(* CODESYS project Struckig_0.17.3.2.library
   Company: Stefan Besler
   DefaultNamespace: Struckig
   Version: 0.17.3.2
   Placeholder: Struckig
   Author: Stefan Besler and contributers
   Description: Full port of pantor ruckig library (Community version) to IEC 61131-3 Structured Text. Online Trajectory Generation. Real-time. Time-optimal. Jerk-constrained.
   Title: Struckig

Project tree, tasks and I/O mapping:
  Struckig/
    _DataTypes/
      data type ControlInterfaceType
      data type DiscretizationType
      data type SynchronizationType
      data type TrajectoryErrorCode
      data type TrajectoryState
    Block/
      data type Block
      data type BlockInterval
    BrakeProfile/
      function block BrakeProfile [ST]: AccelerationBrake, Finalize, FinalizeSecondOrder, PositionBrakeTrajectory, SecondOrderPositionBrakeTrajectory, SecondOrderVelocityBrakeTrajectory, SmoothVelocityBrake, VelocityAtTime, VelocityAtZeroAcceleration, velocityBrake, VelocityBrakeTrajectory
    Math/
      function BubbleSortLreal [ST]
      function Cbrt [ST]
      function Ceil [ST]
      function Clamp [ST]
      function Fmod [ST]
      function IsInfinity [ST]
      function IsNaN [ST]
      function LrealBits [ST]
      function LrealFromBits [ST]
      function Power [ST]
      function Power2 [ST]
      program Roots [ST]: PolyDeri, PolyEval, PolyMonicDeri, ShrinkInterval, SolveCub, SolveQuartMonic, SolveResolvent
    Position/
      function block PositionFirstOrderStep1 [ST]: Get, Set
      function block PositionFirstOrderStep2 [ST]: Get, Set
      function block PositionSecondOrderStep1 [ST]: AddInterval, AddProfile, CalculateBlock, Get, RemoveProfile, Set, time_acc0, time_all_single_step, time_none
      function block PositionSecondOrderStep2 [ST]: CheckAll, Get, Set, time_acc0, time_none
      function block PositionThirdOrderStep1 [ST]: AddInterval, AddProfile, CalculateBlock, Get, RemoveProfile, Set, time_acc0_acc1, time_acc0_two_step, time_acc1_vel_two_step, time_all_none_acc0_acc1, time_all_single_step, time_all_vel, time_none_two_step, time_vel_two_step
      function block PositionThirdOrderStep2 [ST]: Get, Set, time_acc0, time_acc0_acc1, time_acc0_acc1_vel, time_acc0_vel, time_acc1, time_acc1_vel, time_none, time_none_smooth, time_vel
    Profile/
      _DataTypes/
        data type ProfileBound
        data type ProfileControlSigns
        data type ProfileDirection
        data type ReachedLimits
      function block ProfileDesc [ST]: Bound, CheckBound, CheckForFirstOrder, CheckForFirstOrderWithTiming, CheckForFirstOrderWithTiming2, CheckForSecondOrder, CheckForSecondOrderVelocity, CheckForSecondOrderVelocityWithTiming, CheckForSecondOrderVelocityWithTiming2, CheckForSecondOrderWithTiming, CheckForSecondOrderWithTiming2, CheckForVelocity, CheckForVelocityWithTiming, CheckStepForBound, CheckVel, CheckWithTiming, CheckWithTiming2, FirstStateAtPosition, SetBoundary, SetBoundaryPosition, SetBoundaryVelocity
    Velocity/
      function block VelocitySecondOrderStep1 [ST]: Get, Set
      function block VelocitySecondOrderStep2 [ST]: Get, Set
      function block VelocityThirdOrderStep1 [ST]: AddInterval, AddProfile, CalculateBlock, Get, RemoveProfile, Set, time_acc0, time_all_single_step, time_none
      function block VelocityThirdOrderStep2 [ST]: CheckAll, Get, Set, time_acc0, time_none
    function Integrate [ST]
    interface IOtg: AtTime, AtTime1, Cyclic, Duration, ErrorCode, ErrorMessage, PassOutputToInput, Reset, State, ValidateInput
    function block Otg [ST]: AbortErrorId, AtTime, AtTime1, Calculate, Cyclic, Duration, ErrorCode, ErrorMessage, FB_init, HasChanged, IsBlocked, IsInputCollinear, PassOutputToInput, Reset, SetBusy, State, Synchronize, ValidateInput, ValidateInputOrAbort, VelocityAtZero
    function block Otg1 [ST]: AtTime, AtTime1, Cyclic, Duration, ErrorCode, ErrorMessage, FB_init, PassOutputToInput, Reset, State, ValidateInput
  global variables Constants
  global variables ParameterList
*)

// Struckig/_DataTypes/ControlInterfaceType
// Struckig
// Copyright (C) 2022 Stefan Besler

// This program is free software: you can redistribute it and/or modify
// it under the terms of the GNU General Public License as published by
// the Free Software Foundation, either version 3 of the License, or
// (at your option) any later version.

// This program is distributed in the hope that it will be useful,
// but WITHOUT ANY WARRANTY; without even the implied warranty of
// MERCHANTABILITY or FITNESS FOR A PARTICULAR PURPOSE.  See the
// GNU General Public License for more details.
//
// You should have received a copy of the GNU General Public License
// along with THIS PROGRAM.  IF NOT, see <http://www.gnu.org/licenses/>.
{attribute 'qualified_only'}
{attribute 'strict'}
/// Defines the controlled state variables for trajectory generation.
/// The selected mode changes which boundary values and limits are interpreted
/// during validation and profile generation.
TYPE ControlInterfaceType :
(
  Undefined, //< Use global/default configuration.
  Position, //< Full control over position, velocity, and acceleration.
  Velocity //< Controls only velocity and acceleration states.
);
END_TYPE

// Struckig/_DataTypes/DiscretizationType
// Struckig
// Copyright (C) 2022 Stefan Besler

// This program is free software: you can redistribute it and/or modify
// it under the terms of the GNU General Public License as published by
// the Free Software Foundation, either version 3 of the License, or
// (at your option) any later version.

// This program is distributed in the hope that it will be useful,
// but WITHOUT ANY WARRANTY; without even the implied warranty of
// MERCHANTABILITY or FITNESS FOR A PARTICULAR PURPOSE.  See the
// GNU General Public License for more details.
//
// You should have received a copy of the GNU General Public License
// along with THIS PROGRAM.  IF NOT, see <http://www.gnu.org/licenses/>.
{attribute 'qualified_only'}
{attribute 'strict'}
/// Defines whether synchronized trajectory duration is continuous or cycle-discrete.
TYPE DiscretizationType :
(
  Continuous, //< Every synchronization duration is allowed.
  Discrete //< Synchronization duration must be a multiple of cycle time.
);
END_TYPE

// Struckig/_DataTypes/SynchronizationType
// Struckig
// Copyright (C) 2022 Stefan Besler

// This program is free software: you can redistribute it and/or modify
// it under the terms of the GNU General Public License as published by
// the Free Software Foundation, either version 3 of the License, or
// (at your option) any later version.

// This program is distributed in the hope that it will be useful,
// but WITHOUT ANY WARRANTY; without even the implied warranty of
// MERCHANTABILITY or FITNESS FOR A PARTICULAR PURPOSE.  See the
// GNU General Public License for more details.
//
// You should have received a copy of the GNU General Public License
// along with THIS PROGRAM.  IF NOT, see <http://www.gnu.org/licenses/>.
{attribute 'qualified_only'}
{attribute 'strict'}
/// Defines how multiple DoFs are synchronized to a common trajectory timing.
/// This setting is evaluated together with per-axis overrides (`PerDofSynchronization`)
/// in [Otg](xref:Struckig.Otg).
TYPE SynchronizationType :
(
  Undefined, //< Use global/default configuration.
  TimeSync, //< Always synchronize the DoFs to reach the target at the same time (Default)
  TimeIfNecessarySync, //< Synchronize only when necessary (e.g. for non-zero target velocity or acceleration)
  Phase,  //< Phase synchronize the DoFs when this is possible, else fallback to "Time" strategy. Phase synchronization will result a straight-line trajectory
    // PhaseOnly, //< Always phase synchronize the DoFs (even when this is not time-optimal), else returns "ErrorNoPhaseSynchronization". Ruckig will then guarantee a straight-line trajectory
  None //< Calculate every DoF independently
);
END_TYPE

// Struckig/_DataTypes/TrajectoryErrorCode
// Struckig
// Copyright (C) 2022 Stefan Besler

// This program is free software: you can redistribute it and/or modify
// it under the terms of the GNU General Public License as published by
// the Free Software Foundation, either version 3 of the License, or
// (at your option) any later version.

// This program is distributed in the hope that it will be useful,
// but WITHOUT ANY WARRANTY; without even the implied warranty of
// MERCHANTABILITY or FITNESS FOR A PARTICULAR PURPOSE.  See the
// GNU General Public License for more details.
//
// You should have received a copy of the GNU General Public License
// along with THIS PROGRAM.  IF NOT, see <http://www.gnu.org/licenses/>.
{attribute 'qualified_only'}
/// Error codes reported by the trajectory generator.
/// Returned by [ErrorCode](xref:Struckig.IOtg#ErrorCode) and explained by
/// [ErrorMessage](xref:Struckig.IOtg#ErrorMessage).
TYPE TrajectoryErrorCode :
(
  Undefined := 0, //< No error.
  InvalidInput, //< Error in the input parameter
  SynchronizationFailed, //< No valid synchronized profile was found.
  CalculateStep1Failed, //< Profile search in step 1 failed.
  ZeroLimitsConflict, //< Conflicting zero limits prevent profile generation.
  ZeroLimitsConflictInSynchronization //< Zero-limit conflict during multi-DoF synchronization.
);
END_TYPE

// Struckig/_DataTypes/TrajectoryState
// Struckig
// Copyright (C) 2022 Stefan Besler

// This program is free software: you can redistribute it and/or modify
// it under the terms of the GNU General Public License as published by
// the Free Software Foundation, either version 3 of the License, or
// (at your option) any later version.

// This program is distributed in the hope that it will be useful,
// but WITHOUT ANY WARRANTY; without even the implied warranty of
// MERCHANTABILITY or FITNESS FOR A PARTICULAR PURPOSE.  See the
// GNU General Public License for more details.
//
// You should have received a copy of the GNU General Public License
// along with THIS PROGRAM.  IF NOT, see <http://www.gnu.org/licenses/>.
{attribute 'qualified_only'}
{attribute 'strict'}
/// Runtime state of the trajectory generator.
TYPE TrajectoryState :
(
  Undefined, //< State has not been initialized yet.
  
  /// The trajectory has reached its final position. For trajectories with a target velocity or/and a target acceleration
  /// there will still be movement.
  Idle,
  
  /// The trajectory is calculated normally
  Busy,
  
  /// An error occured, use [ErrorCode](xref:Struckig.IOtg#ErrorCode) and [ErrorMessage](xref:Struckig.IOtg#ErrorMessage) to get more
  /// information about the error.
  Error
);
END_TYPE

// Struckig/Block/Block
// Struckig
// Copyright (C) 2022 Stefan Besler

// This program is free software: you can redistribute it and/or modify
// it under the terms of the GNU General Public License as published by
// the Free Software Foundation, either version 3 of the License, or
// (at your option) any later version.

// This program is distributed in the hope that it will be useful,
// but WITHOUT ANY WARRANTY; without even the implied warranty of
// MERCHANTABILITY or FITNESS FOR A PARTICULAR PURPOSE.  See the
// GNU General Public License for more details.
//
// You should have received a copy of the GNU General Public License
// along with THIS PROGRAM.  IF NOT, see <http://www.gnu.org/licenses/>.
TYPE INTERNAL Block :
STRUCT
  Pmin : ProfileDesc; // Save min Profile so that it doesn't need to be recalculated in Step2
  Tmin : LREAL; // [s]
  A, B : BlockInterval; // Max. 2 intervals can be blocked: called a and b with corresponding profiles, order does not matter  
END_STRUCT
END_TYPE

// Struckig/Block/BlockInterval
// Struckig
// Copyright (C) 2022 Stefan Besler

// This program is free software: you can redistribute it and/or modify
// it under the terms of the GNU General Public License as published by
// the Free Software Foundation, either version 3 of the License, or
// (at your option) any later version.

// This program is distributed in the hope that it will be useful,
// but WITHOUT ANY WARRANTY; without even the implied warranty of
// MERCHANTABILITY or FITNESS FOR A PARTICULAR PURPOSE.  See the
// GNU General Public License for more details.
//
// You should have received a copy of the GNU General Public License
// along with THIS PROGRAM.  IF NOT, see <http://www.gnu.org/licenses/>.
/// Which times are possible for synchronization?
TYPE INTERNAL BlockInterval :
STRUCT
  IsUsed : BOOL;
  Left, Right : LREAL;
  Profile : ProfileDesc;
END_STRUCT
END_TYPE

// Struckig/Profile/_DataTypes/ProfileBound
// Struckig
// Copyright (C) 2022 Stefan Besler

// This program is free software: you can redistribute it and/or modify
// it under the terms of the GNU General Public License as published by
// the Free Software Foundation, either version 3 of the License, or
// (at your option) any later version.

// This program is distributed in the hope that it will be useful,
// but WITHOUT ANY WARRANTY; without even the implied warranty of
// MERCHANTABILITY or FITNESS FOR A PARTICULAR PURPOSE.  See the
// GNU General Public License for more details.
//
// You should have received a copy of the GNU General Public License
// along with THIS PROGRAM.  IF NOT, see <http://www.gnu.org/licenses/>.
{attribute 'conditionalshow'}
/// Positional envelope of a single-DoF profile.
/// The structure stores minimum/maximum position and the corresponding
/// times where these extrema occur along the generated trajectory.
///
/// It is returned by profile-bound checks to answer questions such as:
/// "What is the furthest negative/positive excursion and when does it happen?"
TYPE ProfileBound :
STRUCT
  Minimum, Maximum : LREAL; //< Extreme positions reached by the profile.
  Tmin, Tmax : LREAL;  //< Times at which `Minimum` and `Maximum` are reached.
END_STRUCT
END_TYPE

// Struckig/Profile/_DataTypes/ProfileControlSigns
// Struckig
// Copyright (C) 2022 Stefan Besler

// This program is free software: you can redistribute it and/or modify
// it under the terms of the GNU General Public License as published by
// the Free Software Foundation, either version 3 of the License, or
// (at your option) any later version.

// This program is distributed in the hope that it will be useful,
// but WITHOUT ANY WARRANTY; without even the implied warranty of
// MERCHANTABILITY or FITNESS FOR A PARTICULAR PURPOSE.  See the
// GNU General Public License for more details.
//
// You should have received a copy of the GNU General Public License
// along with THIS PROGRAM.  IF NOT, see <http://www.gnu.org/licenses/>.
{attribute 'qualified_only'}
{attribute 'strict'}
TYPE INTERNAL ProfileControlSigns :
(
  Uddu,
  Udud 
);
END_TYPE

// Struckig/Profile/_DataTypes/ProfileDirection
// Struckig
// Copyright (C) 2022 Stefan Besler

// This program is free software: you can redistribute it and/or modify
// it under the terms of the GNU General Public License as published by
// the Free Software Foundation, either version 3 of the License, or
// (at your option) any later version.

// This program is distributed in the hope that it will be useful,
// but WITHOUT ANY WARRANTY; without even the implied warranty of
// MERCHANTABILITY or FITNESS FOR A PARTICULAR PURPOSE.  See the
// GNU General Public License for more details.
//
// You should have received a copy of the GNU General Public License
// along with THIS PROGRAM.  IF NOT, see <http://www.gnu.org/licenses/>.
{attribute 'qualified_only'}
{attribute 'strict'}
TYPE INTERNAL ProfileDirection :
(
  Up,
  Down
);
END_TYPE

// Struckig/Profile/_DataTypes/ReachedLimits
// Struckig
// Copyright (C) 2022 Stefan Besler

// This program is free software: you can redistribute it and/or modify
// it under the terms of the GNU General Public License as published by
// the Free Software Foundation, either version 3 of the License, or
// (at your option) any later version.

// This program is distributed in the hope that it will be useful,
// but WITHOUT ANY WARRANTY; without even the implied warranty of
// MERCHANTABILITY or FITNESS FOR A PARTICULAR PURPOSE.  See the
// GNU General Public License for more details.
//
// You should have received a copy of the GNU General Public License
// along with THIS PROGRAM.  IF NOT, see <http://www.gnu.org/licenses/>.
{attribute 'qualified_only'}
{attribute 'strict'}
TYPE INTERNAL ReachedLimits :
(
  Acc0Acc1Vel,
  Vel, 
  Acc0,
  Acc1,
  Acc0Acc1,
  Acc0Vel,
  Acc1Vel,
  None
);
END_TYPE

// Constants
// Struckig
// Copyright (C) 2022 Stefan Besler

// This program is free software: you can redistribute it and/or modify
// it under the terms of the GNU General Public License as published by
// the Free Software Foundation, either version 3 of the License, or
// (at your option) any later version.

// This program is distributed in the hope that it will be useful,
// but WITHOUT ANY WARRANTY; without even the implied warranty of
// MERCHANTABILITY or FITNESS FOR A PARTICULAR PURPOSE.  See the
// GNU General Public License for more details.
//
// You should have received a copy of the GNU General Public License
// along with THIS PROGRAM.  IF NOT, see <http://www.gnu.org/licenses/>.
{attribute 'qualified_only'}
{attribute 'hide'}
VAR_GLOBAL CONSTANT
  BrakeEpsilon : LREAL := 2.2E-14;
  DoubleEpsilon : LREAL := 2.2204460492503131E-016; // smallest such that 1.0+Constants.DoubleEpsilon != 1.0
  Epsilon : LREAL := 1E-8;
  Epsilon16 : LREAL := 16 * 2.2204460492503131E-016;
  EpsilonColinear : LREAL := 1E-7;
  Infinity : LREAL := 1.7976931348623157E+308;  
  Tolerance : LREAL := 1E-14;
  Cos120 : LREAL := -0.50;
  Sin120 : LREAL := 0.866025403784438646764;  
  Pi : LREAL := 3.14159265358979323846;
  Minimum : LREAL := 1.17549435082E-38;  // used for validating input
  
  VelocityEpsilon : LREAL := 1E-12;
  AccelerationEpsilon : LREAL := 1E-12;
  JerkEpsilon : LREAL := 1E-12; 
  
  PositionPrecision : LREAL := 1E-8;
  VelocityPrecision : LREAL := 1E-8;
  AccelerationPrecision : LREAL := 1E-10;
  TimePrecision : LREAL := 1E-12;  
  
  Tmax : LREAL := 1E12;
END_VAR

// ParameterList
// Struckig
// Copyright (C) 2022 Stefan Besler

// This program is free software: you can redistribute it and/or modify
// it under the terms of the GNU General Public License as published by
// the Free Software Foundation, either version 3 of the License, or
// (at your option) any later version.

// This program is distributed in the hope that it will be useful,
// but WITHOUT ANY WARRANTY; without even the implied warranty of
// MERCHANTABILITY or FITNESS FOR A PARTICULAR PURPOSE.  See the
// GNU General Public License for more details.
//
// You should have received a copy of the GNU General Public License
// along with THIS PROGRAM.  IF NOT, see <http://www.gnu.org/licenses/>.
{attribute 'qualified_only'}
/// Global configuration constants for Struckig.
/// These values define library limits and algorithm defaults that are
/// referenced by trajectory generation and numerical helper routines.
VAR_GLOBAL CONSTANT
  MaxDoFs : INT := 7; //< Maximum number of degrees of freedom supported by `Otg`.
  MaxIterations : BYTE := 127; //< Maximum iterations when [shrinking an interval](xref:Struckig.Roots#ShrinkInterval)
  NumericalRobust : BOOL := TRUE; //< Enables additional guards for numerically robust calculations.
  
  /// Default initial value for Otg.SmoothBrake / Otg1.SmoothBrake
  /// If enabled, braking profiles prefer smooth acceleration transitions.
  SmoothBrake : BOOL := FALSE;
END_VAR

// Struckig/BrakeProfile/BrakeProfile
// Struckig
// Copyright (C) 2022 Stefan Besler

// This program is free software: you can redistribute it and/or modify
// it under the terms of the GNU General Public License as published by
// the Free Software Foundation, either version 3 of the License, or
// (at your option) any later version.

// This program is distributed in the hope that it will be useful,
// but WITHOUT ANY WARRANTY; without even the implied warranty of
// MERCHANTABILITY or FITNESS FOR A PARTICULAR PURPOSE.  See the
// GNU General Public License for more details.
//
// You should have received a copy of the GNU General Public License
// along with THIS PROGRAM.  IF NOT, see <http://www.gnu.org/licenses/>.
/// Calculates (pre- or post-) profile to get current or final state below the limits
FUNCTION_BLOCK BrakeProfile
VAR_INPUT
  Duration : LREAL; //! Overall duration
  t, j, a, v, p : ARRAY[0..2] OF LREAL; //! Profile information for up to three-step profile  
  IsUsed : BOOL;
END_VAR
VAR
  t_to_a_min, t_to_a_max, t_min_to_v_max, t_to_a_zero, t_to_v_min, t_to_v_max : LREAL;
  t_to_v_max_with_constant, t_to_v_min_with_constant, v_at_a0, v_at_a_max, v_at_a_min : LREAL;
END_VAR

METHOD AccelerationBrake
VAR_INPUT
  v0, a0 : LREAL;
  vMax, vMin : LREAL;
  aMax, aMin : LREAL;
  jMax : LREAL;
END_VAR
j[0] := -jMax;

t_to_a_max := (a0 - aMax) / jMax;
t_to_a_zero := a0 / jMax;

v_at_a_max := VelocityAtTime(v0, a0, -jMax, t_to_a_max);
v_at_a0 := VelocityAtTime(v0, a0, -jMax, t_to_a_zero);

IF (v_at_a0 > vMax AND_THEN jMax > 0) OR_ELSE (v_at_a0 < vMax AND_THEN jMax < 0)
THEN
  VelocityBrake(v0, a0, vMax, vMin, aMax, aMin, jMax);

ELSIF (v_at_a_max < vMin AND_THEN jMax > 0) OR_ELSE (v_at_a_max > vMin AND_THEN jMax < 0)
THEN
  t_to_v_min := -(v_at_a_max - vMin)/aMax;
  t_to_v_max := -aMax/(2*jMax) - (v_at_a_max + vMax)/aMax;
  t[0] := t_to_a_max + Constants.BrakeEpsilon;
  t[1] := MAX(MIN(t_to_v_min, v_at_a_max - Constants.BrakeEpsilon), 0.0);
ELSE
  t[0] := t_to_a_max + Constants.BrakeEpsilon;
END_IF
END_METHOD

/// Finalize third-order braking by integrating along kinematic state
METHOD Finalize
VAR_IN_OUT
  ps : LREAL;
  vs : LREAL;
  as : LREAL;
END_VAR
IF t[0] <= 0 AND_THEN t[1] <= 0
THEN
  Duration := 0;
  RETURN;
END_IF

Duration := t[0];
p[0] := ps;
v[0] := vs;
a[0] := as;
Integrate(t[0], p0:=ps, v0:=vs, a0:=as, j:=j[0], p:=ps, v:=vs, a:=as);

IF t[1] > 0
THEN
  Duration := Duration + t[1];
  p[1] := ps;
  v[1] := vs;
  a[1] := as;
  Integrate(t[1], p0:=ps, v0:=vs, a0:=as, j:=j[1], p:=ps, v:=vs, a:=as);
END_IF

IF t[2] > 0
THEN
  Duration := Duration + t[2];
  p[2] := ps;
  v[2] := vs;
  a[2] := as;
  Integrate(t[2], p0:=ps, v0:=vs, a0:=as, j:=j[2], p:=ps, v:=vs, a:=as);
END_IF
END_METHOD

/// Finalize third-order braking by integrating along kinematic state
METHOD FinalizeSecondOrder
VAR_IN_OUT
  ps : LREAL;
  vs : LREAL;
  as : LREAL;
END_VAR
IF t[0] <= 0.0
THEN
  Duration := 0;
  RETURN;
END_IF

Duration := t[0];
p[0] := ps;
v[0] := vs;
Integrate(t[0], p0:=ps, v0:=vs, a0:=a[0], j:=j[0], p:=ps, v:=vs, a:=as);
END_METHOD

/// Calculate brake trajectory for third-order position interface
METHOD PositionBrakeTrajectory
VAR_INPUT
  v0, a0 : LREAL;
  vMax, vMin : LREAL;
  aMax, aMin : LREAL;
  jMax : LREAL;
  SmoothBrake : BOOL;
END_VAR
t[0] := 0.0;
t[1] := 0.0;
t[2] := 0.0;
j[0] := 0.0;
j[1] := 0.0;
j[2] := 0.0;

IF jMax = 0 OR_ELSE aMax = 0 OR_ELSE aMin = 0
THEN
  RETURN;
ELSIF a0 > aMax
THEN
  AccelerationBrake(v0, a0, vMax, vMin, aMax, aMin, jMax);
ELSIF a0 < aMin
THEN
  AccelerationBrake(v0, a0, vMin, vMax, aMin, aMax, -jMax);
ELSIF SmoothBrake AND_THEN v0 > vMax AND_THEN ABS(a0) < aMax
THEN
  SmoothVelocityBrake(v0, a0, vMax, aMax, jMax);
  IF t[0] <= 0 THEN
    VelocityBrake(v0, a0, vMax, vMin, aMax, aMin, jMax);
  END_IF
ELSIF SmoothBrake AND_THEN v0 < vMin AND_THEN ABS(a0) < aMax
THEN
  SmoothVelocityBrake(v0, a0, vMin, aMax, -jMax);
  IF t[0] <= 0 THEN
    VelocityBrake(v0, a0, vMin, vMax, aMin, aMax, -jMax);
  END_IF
ELSIF ((v0 > vMax AND_THEN VelocityAtZeroAcceleration(v0, a0, -jMax) > vMin) OR_ELSE (a0 > 0 AND_THEN VelocityAtZeroAcceleration(v0, a0, jMax) > vMax))
THEN
  VelocityBrake(v0, a0, vMax, vMin, aMax, aMin, jMax);
ELSIF ((v0 < vMin AND_THEN VelocityAtZeroAcceleration(v0, a0, jMax) < vMax) OR_ELSE (a0 < 0 AND_THEN VelocityAtZeroAcceleration(v0, a0, -jMax) < vMin))
THEN
  VelocityBrake(v0, a0, vMin, vMax, aMin, aMax, -jMax);      
END_IF
END_METHOD

/// Calculate brake trajectory for third-order position interface
METHOD SecondOrderPositionBrakeTrajectory
VAR_INPUT
  v0 : LREAL;
  vMax, vMin : LREAL;
  aMax, aMin : LREAL;
END_VAR
t[0] := 0.0;
t[1] := 0.0;
j[0] := 0.0;
j[1] := 0.0;
a[0] := 0.0;
a[1] := 0.0;

IF aMax = 0.0 OR_ELSE aMin = 0.0
THEN
  RETURN; // Ignore braking for zero-limits 
END_IF

IF v0 > vMax
THEN
  a[0] := aMin;
  t[0] := (vMax - v0)/aMin + Constants.Epsilon;   
ELSIF v0 < vMin
THEN
  a[0] := aMax;
  t[0] := (vMin - v0)/aMax + Constants.Epsilon;
END_IF
END_METHOD

/// Calculate brake trajectory for third-order position interface
METHOD SecondOrderVelocityBrakeTrajectory
VAR_INPUT
END_VAR
t[0] := 0;
t[1] := 0;
j[0] := 0;
j[1] := 0;
END_METHOD

/// Jerk-limited brake from (v0, a0) to (vTarget, a=0).
/// Produces a 2- or 3-phase profile that ends with zero acceleration,
/// so Step1 does not inherit a large residual deceleration.
/// jMax > 0 means braking from above (v0 > vTarget), jMax < 0 means from below.
/// If the profile cannot be computed (e.g. a0 opposes braking too strongly),
/// t[0] remains 0 so the caller can fall back to legacy VelocityBrake.
METHOD SmoothVelocityBrake
VAR_INPUT
  v0, a0 : LREAL;
  vTarget : LREAL;
  aMax : LREAL;
  jMax : LREAL;
END_VAR
VAR
  half_D, t1, t3, a_peak : LREAL;
  v1, dv_phase3, t2, a_clamp : LREAL;
END_VAR
IF (jMax > 0 AND_THEN v0 <= vTarget) OR_ELSE (jMax < 0 AND_THEN v0 >= vTarget) THEN
  RETURN;
END_IF

(* Solve quadratic for 2-phase brake from (v0,a0) to (vTarget,0):
   Phase 1: j = -jMax, duration t1
   Phase 3: j = +jMax, duration t3 = t1 - a0/jMax
   jMax * t1^2 - 2*a0*t1 + (vTarget - v0 + a0^2/(2*jMax)) = 0
   D/4 = a0^2/2 + jMax*(v0 - vTarget) *)
half_D := a0*a0*0.5 + jMax*(v0 - vTarget);
IF half_D < 0 THEN
  RETURN;
END_IF

IF jMax > 0 THEN
  t1 := (a0 + SQRT(half_D)) / jMax;
ELSE
  t1 := (a0 - SQRT(half_D)) / jMax;
END_IF

IF t1 < 0 THEN
  RETURN;
END_IF

t3 := t1 - a0/jMax;
a_peak := a0 - jMax*t1;

IF ABS(a_peak) <= aMax THEN
  j[0] := -jMax;
  t[0] := t1;
  j[1] := jMax;
  t[1] := t3;
  t[2] := 0;
ELSE
  (* 3-phase: clamp peak acceleration at ±aMax *)
  IF jMax > 0 THEN
    a_clamp := -aMax;
  ELSE
    a_clamp := aMax;
  END_IF

  t1 := (a0 - a_clamp) / jMax;
  t3 := -a_clamp / jMax;
  v1 := v0 + a0*t1 - 0.5*jMax*t1*t1;
  dv_phase3 := a_clamp*t3 + 0.5*jMax*t3*t3;
  t2 := (vTarget - v1 - dv_phase3) / a_clamp;

  IF t2 < 0 THEN
    RETURN;
  END_IF

  j[0] := -jMax;
  t[0] := t1;
  j[1] := 0;
  t[1] := t2;
  j[2] := jMax;
  t[2] := t3;
END_IF
END_METHOD

METHOD VelocityAtTime : LREAL
VAR_INPUT
  v0, a0 : LREAL;
  j : LREAL;
  t : LREAL;
END_VAR
VelocityAtTime := v0 + t * (a0 + j * t * 0.5);
END_METHOD

METHOD VelocityAtZeroAcceleration : LREAL
VAR_INPUT
  v0, a0 : LREAL;
  j : LREAL;
END_VAR
VelocityAtZeroAcceleration := v0 + (a0 * a0) / (2 * j);
END_METHOD

METHOD VelocityBrake
VAR_INPUT
  v0, a0 : LREAL;
  vMax, vMin : LREAL;
  aMax, aMin : LREAL;
  jMax : LREAL;
END_VAR
j[0] := -jMax;
t_to_a_min := (a0 - aMin)/jMax;
t_to_v_max := a0*a0 + 2 * jMax * (v0 - vMax);
t_to_v_min := a0*a0 / 2 + jMax * (v0 - vMin);

IF t_to_v_max < 0 OR_ELSE t_to_v_min < 0
THEN
  RETURN;
END_IF

t_to_v_max := a0/jMax + SQRT(t_to_v_max) / ABS(jMax);
t_to_v_min := a0/jMax + SQRT(t_to_v_min) / ABS(jMax);
t_min_to_v_max := MIN(t_to_v_max, t_to_v_min);

IF (t_to_a_min < t_min_to_v_max)
THEN
  v_at_a_min := VelocityAtTime(v0, a0, -jMax, t_to_a_min);
  t_to_v_max_with_constant := -(v_at_a_min - vMax)/aMin;
  t_to_v_min_with_constant := -0.5*aMin/jMax - (v_at_a_min - vMin)/aMin;
  t[0] := MAX(t_to_a_min - Constants.BrakeEpsilon, 0);
  t[1] := MAX(MIN(t_to_v_max_with_constant, t_to_v_min_with_constant), 0.0);
ELSE
  t[0] := MAX(t_min_to_v_max - Constants.BrakeEpsilon, 0);
END_IF
END_METHOD

/// Calculate brake trajectory for third-order velocity interface
METHOD VelocityBrakeTrajectory
VAR_INPUT
  v0, a0 : LREAL;
  aMax, aMin : LREAL;
  jMax : LREAL;
END_VAR
t[0] := 0.0;
t[1] := 0.0;
j[0] := 0.0;
j[1] := 0.0;

IF jMax = 0
THEN
  RETURN; // Ignore braking for zero-limits
ELSIF (a0 > aMax)
THEN
  j[0] := -jMax;
  t[0] := (a0 - aMax)/jMax + Constants.BrakeEpsilon;
ELSIF (a0 < aMin)
THEN
  j[0] := jMax;
  t[0] := -(a0 - aMin)/jMax + Constants.BrakeEpsilon;
END_IF
END_METHOD

END_FUNCTION_BLOCK

// Struckig/Integrate
// Struckig
// Copyright (C) 2022 Stefan Besler

// This program is free software: you can redistribute it and/or modify
// it under the terms of the GNU General Public License as published by
// the Free Software Foundation, either version 3 of the License, or
// (at your option) any later version.

// This program is distributed in the hope that it will be useful,
// but WITHOUT ANY WARRANTY; without even the implied warranty of
// MERCHANTABILITY or FITNESS FOR A PARTICULAR PURPOSE.  See the
// GNU General Public License for more details.
//
// You should have received a copy of the GNU General Public License
// along with THIS PROGRAM.  IF NOT, see <http://www.gnu.org/licenses/>.
/// Integrate with constant jerk for duration t. Returns new position, new velocity, and new acceleration.
FUNCTION INTERNAL Integrate
VAR_INPUT
  t, p0, v0, a0, j : LREAL;
END_VAR
VAR_IN_OUT
  p, v, a : LREAL;
END_VAR

p := p0 + t * (v0 + t * (a0 * 0.5 + t * j / 6));
v := v0 + t * (a0 + t * j * 0.5);
a := a0 + t * j;

END_FUNCTION

// Struckig/Math/Clamp
// Struckig
// Copyright (C) 2022 Stefan Besler

// This program is free software: you can redistribute it and/or modify
// it under the terms of the GNU General Public License as published by
// the Free Software Foundation, either version 3 of the License, or
// (at your option) any later version.

// This program is distributed in the hope that it will be useful,
// but WITHOUT ANY WARRANTY; without even the implied warranty of
// MERCHANTABILITY or FITNESS FOR A PARTICULAR PURPOSE.  See the
// GNU General Public License for more details.
//
// You should have received a copy of the GNU General Public License
// along with THIS PROGRAM.  IF NOT, see <http://www.gnu.org/licenses/>.
/// Clamps `value` to the closed interval `[minimum, maximum]`.
/// If `value` is below `minimum`, returns `minimum`.
/// If `value` is above `maximum`, returns `maximum`.
FUNCTION Clamp : LREAL
VAR_INPUT
  value : LREAL; //< Input value to clamp.
  minimum : LREAL; //< Lower bound.
  maximum : LREAL; //< Upper bound.
END_VAR

Clamp := MIN(MAX(value, minimum), maximum);

END_FUNCTION

// Struckig/Math/BubbleSortLreal
// Struckig
// Copyright (C) 2022 Stefan Besler

// This program is free software: you can redistribute it and/or modify
// it under the terms of the GNU General Public License as published by
// the Free Software Foundation, either version 3 of the License, or
// (at your option) any later version.

// This program is distributed in the hope that it will be useful,
// but WITHOUT ANY WARRANTY; without even the implied warranty of
// MERCHANTABILITY or FITNESS FOR A PARTICULAR PURPOSE.  See the
// GNU General Public License for more details.
//
// You should have received a copy of the GNU General Public License
// along with THIS PROGRAM.  IF NOT, see <http://www.gnu.org/licenses/>.
{attribute 'hide'}
/// Internal bubble-sort helper for `LREAL` arrays.
/// Returns sorted index positions in `indicesSorted` without modifying input `data`.
FUNCTION BubbleSortLreal : BOOL
VAR_INPUT
  data : POINTER TO LREAL; //< Input unsorted array.
  size : INT; //< Number of elements in `data`.
  indicesSorted : POINTER TO INT; //< Output sorted indices.
END_VAR
VAR
  i, j, h : INT;
END_VAR

FOR i:=0 TO size
DO
  indicesSorted[i] := i;
END_FOR

// Bubblesort possible_t_syncs from best to worst
FOR i:=0 TO size-1
DO
  FOR j:=0 TO size-1-i
  DO  
    IF data[indicesSorted[j]] > data[indicesSorted[j+1]]
    THEN
      h := indicesSorted[j];
      indicesSorted[j] := indicesSorted[j+1];
      indicesSorted[j+1] := h;     
		END_IF
  END_FOR
END_FOR

END_FUNCTION

// Struckig/Math/Cbrt
// Struckig
// Copyright (C) 2022 Stefan Besler

// This program is free software: you can redistribute it and/or modify
// it under the terms of the GNU General Public License as published by
// the Free Software Foundation, either version 3 of the License, or
// (at your option) any later version.

// This program is distributed in the hope that it will be useful,
// but WITHOUT ANY WARRANTY; without even the implied warranty of
// MERCHANTABILITY or FITNESS FOR A PARTICULAR PURPOSE.  See the
// GNU General Public License for more details.
//
// You should have received a copy of the GNU General Public License
// along with THIS PROGRAM.  IF NOT, see <http://www.gnu.org/licenses/>.
/// The TwinCAT code is a modified version of the original C code from
/// http://www.netlib.org/fdlibm/s_cbrt.c and came with this notice.
///
/// ```
/// Copyright (C) 1993 by Sun Microsystems, Inc. All rights reserved.
///
/// Developed at SunSoft, a Sun Microsystems, Inc. business.
/// Permission to use, copy, modify, and distribute this
/// software is freely granted, provided that this notice
/// is preserved.
/// ```
///
///
/// Small modifications were made, while the original code said
/// ```
/// chop to 20 bits, make larger than cbrt(x)
/// t := LrealFromBits((LrealBits(t) AND SHL(H, 28)) + SHL(J, 30));
/// ```
/// Modern compilers seem to round t away from 0 to 23 bits.
/// see https://github.com/stdlib-js/math-base-special-cbrt/blob/main/src/cbrt.c
{attribute 'hide'}
FUNCTION Cbrt : LREAL
VAR_INPUT
  x : LREAL;
END_VAR
VAR CONSTANT
  B1 : ULINT := 715094163;                  // (682-0.03306235651)*2**20
  B2 : ULINT := 696219795;                  // (664-0.03306235651)*2**20
  C : LREAL := 5.42857142857142815906E-01;  // 19/35     = 0x3FE15F15F15F15F1
  D : LREAL := -7.05306122448979611050E-01; // -864/1225 = 0xBFE691DE2532C834
  E : LREAL := 1.41428571428571436819E+00;  // 99/70     = 0x3FF6A0EA0EA0EA0F
  F : LREAL := 1.60714285714285720630E+00;  // 45/28     = 0x3FF9B6DB6DB6DB6E
  G : LREAL := 3.57142857142857150787E-01;  // 5/14      = 0x3FD6DB6DB6DB6DB7
  J : ULINT := 1;
  Mask : ULINT := ULINT#16#FFFFFFFFC0000000;
  AMask : ULINT := ULINT#16#80000000;
  SmallestNormal : LREAL := 2.22507385850720138309E-308; // 2**-1022  = 0x0010000000000000  
END_VAR
VAR
  sign : BOOL;
  t, r1, s1, w : LREAL;
END_VAR

// test x=0 and x=NaN
IF x = 0 OR_ELSE x <> x
THEN
  Cbrt := x;
  RETURN;
END_IF

sign := FALSE;
IF x < 0
THEN
  x := -x;
  sign := TRUE;  
END_IF

// rough cbrt to 5 bits
t := LrealFromBits(LrealBits(x)/3 + SHL(B1, 32));
IF x < SmallestNormal
THEN
  // subnormal number
  t := LrealFromBits(SHL(J, 54)); // set t= 2**54
  t := t * x;
  t := LrealFromBits(LrealBits(t)/3 + SHL(B2, 32));
END_IF

// new cbrt to 23 bits
r1 := t * t / x;
s1 := C + r1*t;
t := t * (G + F/(s1+E+D/s1));

// see https://github.com/stdlib-js/math-base-special-cbrt/blob/main/src/cbrt.c
t := LrealFromBits((LrealBits(t) + AMask) AND Mask);

// one step newton iteration to 53 bits with error less than 0.667ulps
s1 := t * t; // t*t is exact
r1 := x / s1;
w := t + t;
r1 := (r1 - t) / (w + r1); // r-s is exact
t := t + t*r1;

// restore the sign bit
IF sign
THEN
  t := -t;
END_IF

Cbrt := t;
    
// this one is a bit more prone to numerical errors
// Cbrt := SEL(x < 0, 1.0, -1.0) * EXPT(ABS(x), 1.0 / 3.0);

END_FUNCTION

// Struckig/Math/LrealFromBits
// Struckig
// Copyright (C) 2022 Stefan Besler

// This program is free software: you can redistribute it and/or modify
// it under the terms of the GNU General Public License as published by
// the Free Software Foundation, either version 3 of the License, or
// (at your option) any later version.

// This program is distributed in the hope that it will be useful,
// but WITHOUT ANY WARRANTY; without even the implied warranty of
// MERCHANTABILITY or FITNESS FOR A PARTICULAR PURPOSE.  See the
// GNU General Public License for more details.
//
// You should have received a copy of the GNU General Public License
// along with THIS PROGRAM.  IF NOT, see <http://www.gnu.org/licenses/>.
{attribute 'hide'}
/// Internal bit-cast helper from raw IEEE-754 bits to `LREAL`.
FUNCTION LrealFromBits : LREAL
VAR_INPUT
  b : ULINT; //< Raw floating-point bit pattern.
END_VAR
VAR
  x : POINTER TO LREAL := ADR(b);
END_VAR

LrealFromBits := x^;

END_FUNCTION

// Struckig/Math/LrealBits
// Struckig
// Copyright (C) 2022 Stefan Besler

// This program is free software: you can redistribute it and/or modify
// it under the terms of the GNU General Public License as published by
// the Free Software Foundation, either version 3 of the License, or
// (at your option) any later version.

// This program is distributed in the hope that it will be useful,
// but WITHOUT ANY WARRANTY; without even the implied warranty of
// MERCHANTABILITY or FITNESS FOR A PARTICULAR PURPOSE.  See the
// GNU General Public License for more details.
//
// You should have received a copy of the GNU General Public License
// along with THIS PROGRAM.  IF NOT, see <http://www.gnu.org/licenses/>.
{attribute 'hide'}
/// Internal bit-cast helper from `LREAL` to raw IEEE-754 bits.
FUNCTION LrealBits : ULINT
VAR_INPUT
  x : LREAL; //< Input floating-point value.
END_VAR
VAR
  b : POINTER TO ULINT := ADR(x);
END_VAR

LrealBits := b^;

END_FUNCTION

// Struckig/Math/Ceil
// Struckig
// Copyright (C) 2022 Stefan Besler

// This program is free software: you can redistribute it and/or modify
// it under the terms of the GNU General Public License as published by
// the Free Software Foundation, either version 3 of the License, or
// (at your option) any later version.

// This program is distributed in the hope that it will be useful,
// but WITHOUT ANY WARRANTY; without even the implied warranty of
// MERCHANTABILITY or FITNESS FOR A PARTICULAR PURPOSE.  See the
// GNU General Public License for more details.
//
// You should have received a copy of the GNU General Public License
// along with THIS PROGRAM.  IF NOT, see <http://www.gnu.org/licenses/>.
/// Returns the smallest integer value greater than or equal to `val`.
/// NaN and +/-Infinity are passed through unchanged.
FUNCTION Ceil : LREAL
VAR_INPUT
  val : LREAL; //< Input value.
END_VAR
VAR CONSTANT
  InfinityBits : ULINT := ULINT#16#7FF0000000000000;
END_VAR
VAR
  InfinityPtr : POINTER TO LREAL := ADR(InfinityBits);
END_VAR

IF val <> val OR_ELSE val = InfinityPtr^ OR_ELSE val = -InfinityPtr^ // nan or inf
THEN
  RETURN;
END_IF

Ceil := DINT_TO_LREAL(LREAL_TO_DINT(val));
IF Ceil < val THEN
	Ceil := Ceil + 1;
END_IF;

END_FUNCTION

// Struckig/Math/Fmod
// Struckig
// Copyright (C) 2022 Stefan Besler

// This program is free software: you can redistribute it and/or modify
// it under the terms of the GNU General Public License as published by
// the Free Software Foundation, either version 3 of the License, or
// (at your option) any later version.

// This program is distributed in the hope that it will be useful,
// but WITHOUT ANY WARRANTY; without even the implied warranty of
// MERCHANTABILITY or FITNESS FOR A PARTICULAR PURPOSE.  See the
// GNU General Public License for more details.
//
// You should have received a copy of the GNU General Public License
// along with THIS PROGRAM.  IF NOT, see <http://www.gnu.org/licenses/>.
/// Floating-point remainder operation.
/// Returns the remainder of `x / y` with truncation toward zero:
/// `x - TRUNC(x / y) * y`.
FUNCTION Fmod : LREAL
VAR_INPUT
  x : LREAL; //< Dividend.
  y : LREAL; //< Divisor.
END_VAR

Fmod := x - TRUNC(x / y) * y;

END_FUNCTION

// Struckig/Math/IsInfinity
// Struckig
// Copyright (C) 2022 Stefan Besler

// This program is free software: you can redistribute it and/or modify
// it under the terms of the GNU General Public License as published by
// the Free Software Foundation, either version 3 of the License, or
// (at your option) any later version.

// This program is distributed in the hope that it will be useful,
// but WITHOUT ANY WARRANTY; without even the implied warranty of
// MERCHANTABILITY or FITNESS FOR A PARTICULAR PURPOSE.  See the
// GNU General Public License for more details.
//
// You should have received a copy of the GNU General Public License
// along with THIS PROGRAM.  IF NOT, see <http://www.gnu.org/licenses/>.
/// Checks whether a floating-point value is positive or negative infinity.
FUNCTION IsInfinity : BOOL
VAR_INPUT
  value : LREAL; //< Input value.
END_VAR

IsInfinity := value = Constants.Infinity OR_ELSE value = -Constants.Infinity;

END_FUNCTION

// Struckig/Math/IsNaN
// Struckig
// Copyright (C) 2022 Stefan Besler

// This program is free software: you can redistribute it and/or modify
// it under the terms of the GNU General Public License as published by
// the Free Software Foundation, either version 3 of the License, or
// (at your option) any later version.

// This program is distributed in the hope that it will be useful,
// but WITHOUT ANY WARRANTY; without even the implied warranty of
// MERCHANTABILITY or FITNESS FOR A PARTICULAR PURPOSE.  See the
// GNU General Public License for more details.
//
// You should have received a copy of the GNU General Public License
// along with THIS PROGRAM.  IF NOT, see <http://www.gnu.org/licenses/>.
/// Checks whether a floating-point value is NaN.
/// Uses the IEEE-754 property that NaN is not equal to itself.
FUNCTION IsNaN : BOOL
VAR_INPUT
  value : LREAL; //< Input value.
END_VAR

IsNaN := value <> value;

END_FUNCTION

// Struckig/Math/Power
// Struckig
// Copyright (C) 2022 Stefan Besler

// This program is free software: you can redistribute it and/or modify
// it under the terms of the GNU General Public License as published by
// the Free Software Foundation, either version 3 of the License, or
// (at your option) any later version.

// This program is distributed in the hope that it will be useful,
// but WITHOUT ANY WARRANTY; without even the implied warranty of
// MERCHANTABILITY or FITNESS FOR A PARTICULAR PURPOSE.  See the
// GNU General Public License for more details.
//
// You should have received a copy of the GNU General Public License
// along with THIS PROGRAM.  IF NOT, see <http://www.gnu.org/licenses/>.
/// Internal power helper that preserves sign for negative bases.
/// Evaluates `sign(v) * |v|^e`.
FUNCTION INTERNAL Power : LREAL
VAR_INPUT
  v : LREAL; //< Base value.
  e : LREAL; //< Exponent.
END_VAR

Power := SEL(v < 0, 1.0, -1.0) * EXPT(ABS(v), e);

END_FUNCTION

// Struckig/Math/Power2
// Struckig
// Copyright (C) 2022 Stefan Besler

// This program is free software: you can redistribute it and/or modify
// it under the terms of the GNU General Public License as published by
// the Free Software Foundation, either version 3 of the License, or
// (at your option) any later version.

// This program is distributed in the hope that it will be useful,
// but WITHOUT ANY WARRANTY; without even the implied warranty of
// MERCHANTABILITY or FITNESS FOR A PARTICULAR PURPOSE.  See the
// GNU General Public License for more details.
//
// You should have received a copy of the GNU General Public License
// along with THIS PROGRAM.  IF NOT, see <http://www.gnu.org/licenses/>.
/// Internal square helper.
/// Returns `v * v`.
FUNCTION INTERNAL Power2 : LREAL
VAR_INPUT
  v : LREAL; //< Input value.
END_VAR

Power2 := v*v;

END_FUNCTION

// Struckig/Math/Roots
// Struckig
// Copyright (C) 2022 Stefan Besler

// This program is free software: you can redistribute it and/or modify
// it under the terms of the GNU General Public License as published by
// the Free Software Foundation, either version 3 of the License, or
// (at your option) any later version.

// This program is distributed in the hope that it will be useful,
// but WITHOUT ANY WARRANTY; without even the implied warranty of
// MERCHANTABILITY or FITNESS FOR A PARTICULAR PURPOSE.  See the
// GNU General Public License for more details.
//
// You should have received a copy of the GNU General Public License
// along with THIS PROGRAM.  IF NOT, see <http://www.gnu.org/licenses/>.
PROGRAM INTERNAL Roots
VAR
  a2, q, qsqrt, r2, q3, aa, t : LREAL;
  a, b, c, d, rr, theta, ux, uyi, inva, invaa, bb, bover3a, p, halfq, yy, inv2b, x, y, uuu, vvv, www, w, h : LREAL;
  discriminant : LREAL;
  e0, e1, q1, q2, p1, p2, dd, sqrtD  : LREAL;
  a3, b3, c3 : LREAL;
  x3 : ARRAY[0..2] OF LREAL;
  number_zeroes : INT;  
  deriv : ARRAY[0 .. 10] OF LREAL;
  fl, fh, temp : LREAL;
  dxold, dx, f,df : LREAL;
  j : INT;
  xn : LREAL;
  iterations : BYTE;
END_VAR

METHOD PolyDeri
VAR_INPUT
  coeffs : POINTER TO LREAL;
  coeffsCount : BYTE;
  out : POINTER TO LREAL;
END_VAR
FOR j:=0 TO coeffsCount DO
  out[j] := (coeffsCount - j) * coeffs[j];
END_FOR
END_METHOD

METHOD PolyEval : LREAL;
VAR_INPUT
  polynom : POINTER TO LREAL;
  degree : INT;
  x : LREAL;
END_VAR
IF degree = 0
THEN
  RETURN;
END_IF

IF (ABS(x) < Constants.DoubleEpsilon) THEN
    PolyEval := polynom[degree];
ELSIF x = 1.0 THEN
  FOR j:= degree TO 0 BY -1
  DO
    PolyEval := PolyEval + polynom[j];
  END_FOR
ELSE
  xn := 1.0;
  FOR j:= degree TO 0 BY -1 
  DO
    PolyEval := PolyEval + polynom[j] * xn;
    xn := xn * x;
  END_FOR
END_IF
END_METHOD

METHOD PolyMonicDeri
VAR_INPUT
  monic_coeffs : POINTER TO LREAL;
  coeffsCount : BYTE;
  out : POINTER TO LREAL;  
END_VAR
VAR
  i : BYTE;
END_VAR
out[0] := 1.0;
FOR i:=1 TO coeffsCount-1 DO
  out[i] := (coeffsCount- i) * (monic_coeffs[i] / (coeffsCount));
END_FOR
END_METHOD

// Calculate a single zero of polynom p(x) inside [lbound, ubound]
// Requirements: p(lbound)*p(ubound) < 0, lbound < ubound
METHOD ShrinkInterval : LREAL
VAR_INPUT
  p : POINTER TO LREAL;
  degree : BYTE;  
  l, h : LREAL;
END_VAR
fl := PolyEval(p, degree, l);
fh := PolyEval(p, degree, h);
IF (fl = 0.0) THEN
  ShrinkInterval := l;
  RETURN;
END_IF

IF (fh = 0.0) THEN
  ShrinkInterval := h;
  RETURN;
END_IF

IF (fl > 0.0)
THEN
  // swap l and h
  temp := l;
  l := h;
  h := temp;
END_IF

ShrinkInterval := (l + h) / 2;
dxold := ABS(h - l);
dx := dxold;
PolyDeri(p, degree, out:=ADR(deriv));
f := PolyEval(p, degree, ShrinkInterval);
df := PolyEval(ADR(deriv), degree-1, ShrinkInterval);
FOR iterations:=0 TO ParameterList.MaxIterations DO
  IF ((((ShrinkInterval - h) * df - f) * ((ShrinkInterval - l) * df - f) > 0.0) OR_ELSE (ABS(2 * f) > ABS(dxold * df))) THEN
    dxold := dx;
    dx := (h - l) / 2;
    ShrinkInterval := l + dx;
    IF (l = ShrinkInterval) THEN
      RETURN;
    END_IF
  ELSE
  
    IF ABS(df) < Constants.Epsilon
    THEN
      dxold := dx;
      dx := (h - l) / 2;
      ShrinkInterval := l + dx;
      IF (l = ShrinkInterval) THEN
        RETURN;
      END_IF
    ELSE
      dxold := dx;
      dx := f / df;
      temp := ShrinkInterval;
      ShrinkInterval := ShrinkInterval - dx;
      IF (temp = ShrinkInterval) THEN
        RETURN;
      END_IF
    END_IF
  END_IF
  
  IF (ABS(dx) < Constants.Tolerance) THEN
    RETURN;
  END_IF
  
  f := PolyEval(p, degree, ShrinkInterval);
  df := PolyEval(ADR(deriv), degree-1, ShrinkInterval);
  IF (f < 0.0) THEN
    l := ShrinkInterval;
  ELSE
    h := ShrinkInterval;
  END_IF
END_FOR
END_METHOD

METHOD SolveCub
VAR_INPUT
  polynom : POINTER TO LREAL;
END_VAR
VAR_IN_OUT
  rootCount : INT;
  roots : ARRAY[0..6] OF LREAL;
END_VAR
rootCount := -1;
a := polynom[0];
b := polynom[1];
c := polynom[2];
d := polynom[3];

IF (ABS(d) < Constants.DoubleEpsilon)
THEN
  // First solution is x = 0
  roots[0] := 0.0;
  rootCount := 1;
  
  // Converting to a quadratic equation
  d := c;
  c := b;
  b := a;
  a := 0.0;
END_IF

IF (ABS(a) < Constants.DoubleEpsilon)
THEN
  IF (ABS(b) < Constants.DoubleEpsilon)
  THEN
    IF ABS(c) > Constants.DoubleEpsilon
    THEN
      // Linear equation
      h := (-d / c);
      IF ABS(c) > Constants.DoubleEpsilon AND_THEN h >= 0
      THEN
        roots[rootCount+1] := h;
        rootCount := rootCount + 1;
      END_IF
    END_IF    
  ELSE
    // Quadratic equation
    discriminant := c * c - 4 * b * d;
    IF discriminant >= 0 AND_THEN ABS(b) > Constants.DoubleEpsilon
    THEN
      inv2b := 1.0 / (2 * b);
      y := SQRT(discriminant);
      
      h := ((-c + y) * inv2b);
      IF h >= 0
      THEN
        roots[rootCount+1] := h;
        rootCount := rootCount + 1;
			END_IF
      
      h := ((-c - y) * inv2b);
      IF h >= 0
      THEN      
        roots[rootCount+1] := ((-c - y) * inv2b);
        rootCount := rootCount + 1;
      END_IF
      
    END_IF
  END_IF

ELSE
  
  // Cubic equation
  inva := 1.0 / a;
  invaa := inva * inva;
  bb := b * b;
  bover3a := b * inva / 3;
  p := (a * c - bb / 3) * invaa;
  halfq := (2 * bb * b - 9 * a * b * c + 27 * a * a * d) / 54 * invaa * inva;
  yy := p * p * p / 27 + halfq * halfq;  
    
  IF (yy > Constants.DoubleEpsilon) THEN
    // Sqrt is positive: one real solution}
    y := SQRT(yy);
    uuu := -halfq + y;
    vvv := -halfq - y;
    www := SEL(ABS(uuu) > ABS(vvv), vvv, uuu);
    w := cbrt(www);
    
    h := (w - p / (3 * w) - bover3a);
    IF h >= 0
    THEN
      roots[rootCount+1] := h;
      rootCount := rootCount + 1;    
		END_IF

  ELSIF (yy < -Constants.DoubleEpsilon) THEN
    // Sqrt is negative: three real solutions
    x := -halfq;
    y := SQRT(-yy);

    // Convert to polar form}
    IF ABS(x) > Constants.DoubleEpsilon THEN
      theta := SEL((x > 0.0), (ATAN(y / x) + Constants.Pi), ATAN(y / x));
      rr := SQRT(x * x - yy);
    ELSE
      // Vertical line}
      theta := Constants.Pi / 2;
      rr := y;
    END_IF
    
    // Calculate cube root
    theta := theta / 3;
    rr := 2 * cbrt(rr);
    // Convert to complex coordinate
    ux := COS(theta) * rr;
    uyi := SIN(theta) * rr;
    // First solution
    h := (ux - bover3a);
    IF h >= 0
    THEN
      roots[rootCount+1] := h;
      rootCount := rootCount + 1;
		END_IF
    
    // Second solution, rotate +120 degrees
    h := ux * Constants.Cos120 - uyi * Constants.Sin120 - bover3a;
    IF h >= 0
    THEN
      roots[rootCount+1] := h;
      rootCount := rootCount + 1;
		END_IF
    
    // Third solution, rotate -120 degrees
    h := ux * Constants.Cos120 + uyi * Constants.Sin120 - bover3a;
    IF h >= 0
    THEN
      roots[rootCount+1] := h;
      rootCount := rootCount + 1;
		END_IF
  ELSE
    // Sqrt is zero: two real solutions
    www := -halfq;
    w := 2 * cbrt(www);
    // First solution
    h := (w - bover3a);
    IF h >= 0
    THEN
      roots[rootCount+1] := h;
      rootCount := rootCount + 1;
		END_IF
    
    // Second solution, rotate +120 degrees
    h := (w * Constants.Cos120 - bover3a);
    IF h >= 0
    THEN
      roots[rootCount+1] := h;
      rootCount := rootCount + 1;
		END_IF
  END_IF
END_IF
END_METHOD

/// Calculate all roots of the monic quartic equation: x^4 + a*x^3 + b*x^2 + c*x + d = 0
METHOD SolveQuartMonic
VAR_INPUT
  polynom : POINTER TO LREAL;  
  degree : LREAL;
END_VAR
VAR_IN_OUT
  rootCount : INT;
  roots : ARRAY[0..6] OF LREAL;
END_VAR
rootCount := -1;

a := polynom[0];
b := polynom[1];
c := polynom[2];
d := polynom[3];
e0 := cbrt(c * c);
IF ABS(d) < Constants.DoubleEpsilon
THEN
  IF ABS(c) < Constants.DoubleEpsilon
  THEN
    roots[rootCount+1] := 0;
    rootCount := rootCount + 1;    

    dd := a * a - 4 * b;
    IF ABS(dd) < Constants.DoubleEpsilon 
    THEN
      roots[rootCount+1] := -a / 2;
      rootCount := rootCount + 1;          
     ELSIF (dd > 0)
     THEN 
      sqrtD := SQRT(dd);
      roots[rootCount+1] := (-a - sqrtD) / 2;
      roots[rootCount+2] := (-a + sqrtD) / 2;
      rootCount := rootCount + 2;       
    END_IF
    RETURN;
  END_IF
  
  IF ABS(a) < Constants.DoubleEpsilon AND_THEN ABS(b) < Constants.DoubleEpsilon
  THEN
    roots[rootCount+1] := 0;
    roots[rootCount+2] := -Cbrt(c);
    rootCount := rootCount + 2;
    RETURN;
  END_IF
END_IF

a3 := -b;
b3 := a * c - 4 * d;
c3 := -a * a * d - c * c + 4 * b * d;

number_zeroes := SolveResolvent(ADR(x3), a3, b3, c3);

y := x3[0];
// Choosing Y with maximal absolute value.
IF (number_zeroes <> 1)
THEN
  IF ABS(x3[1]) > ABS(y)
  THEN
    y := x3[1];
  END_IF
  
  IF ABS(x3[2]) > ABS(y)
  THEN
    y := x3[2];
  END_IF
END_IF

// h1 + h2 = y AND_THEN h1*h2 = d  <=>  h^2 - y*h + d = 0    (h === q)
dd := y * y - 4 * d;
IF (ABS(dd) < Constants.DoubleEpsilon) THEN
  q1 := q2 := y / 2;
  // g1 + g2 = a AND_THEN g1 + g2 = b - y   <=>   g^2 - a*g + b - y = 0    (p === g)}
  dd := a * a - 4 * (b - y);
  IF (ABS(dd) < Constants.DoubleEpsilon) THEN
    p1 := p2 := a / 2;
  ELSE
    
    IF dd < 0
    THEN
      RETURN;
    END_IF
    
    sqrtD := SQRT(dd);
    p1 := (a + sqrtD) / 2;
    p2 := (a - sqrtD) / 2;
  END_IF
ELSE
  IF dd < 0
  THEN
    RETURN;
  END_IF
	
  sqrtD := SQRT(dd);
  q1 := (y + sqrtD) / 2;
  q2 := (y - sqrtD) / 2;
  // g1 + g2 = a AND_THEN g1*h2 + g2*h1 = c   ( AND_THEN g === p )  Krammer
  
  IF ABS(q1 - q2) < Constants.DoubleEpsilon
  THEN
    RETURN;
  END_IF
  
  p1 := (a * q1 - c) / (q1 - q2);
  p2 := (c - a * q2) / (q1 - q2);
END_IF

// Solve the quadratic equation: x^2 + p1*x + q1 = 0
dd := p1 * p1 - 4 * q1;
IF ABS(dd) < Constants.Epsilon16
THEN
  
  h:= (-p1 / 2);
  IF h >= 0
  THEN
    roots[rootCount+1] := h;
    rootCount := rootCount + 1;
  END_IF
  
ELSIF dd > 0.0
THEN
  sqrtD := SQRT(dd);
  h := ((-p1 + sqrtD) / 2);
  IF h >= 0
  THEN
    roots[rootCount+1] := h;
    rootCount := rootCount + 1;
  END_IF
    
  h := ((-p1 - sqrtD) / 2);
  IF h >= 0
  THEN
    roots[rootCount+1] := h;
    rootCount := rootCount + 1;
  END_IF
END_IF

// Solve the quadratic equation: x^2 + p2*x + q2 = 0
dd := p2 * p2 - 4 * q2;
IF (ABS(dd) < Constants.Epsilon16) THEN
  h := (-p2 * 0.5);
  IF h >= 0
  THEN
    roots[rootCount+1] := h;
    rootCount := rootCount + 1;
  END_IF  
ELSIF (dd > 0.0) THEN
  sqrtD := SQRT(dd);
  
  h := ((-p2 - sqrtD) / 2);
  IF h >= 0
  THEN
    roots[rootCount+1] := h;
    rootCount := rootCount + 1;
  END_IF
  
  h := ((-p2 + sqrtD) / 2); 
  IF h >= 0
  THEN
    roots[rootCount+1] := h;
    rootCount := rootCount + 1;
  END_IF
END_IF
END_METHOD

/// Solve resolvent eqaution of corresponding Quartic equation
/// The input x must be of length 3
/// Number of zeros are returned
METHOD SolveResolvent : INT
VAR_INPUT
  x : POINTER TO LREAL;
  a,b,c : LREAL;
END_VAR
a := a / 3;
a2 := a * a;
q := a2 - b / 3;
rr := (a * (2 * a2 - b) + c) / 2;
r2 := rr * rr;
q3 := q * q * q;

IF (r2 < q3) AND_THEN q >= 0 THEN
  qsqrt := SQRT(q);
  t := Clamp(rr / (q * qsqrt), -1.0, 1.0);
  q := -2 * SQRT(q);
  theta := ACOS(t) / 3;
  ux := COS(theta) * q;
  uyi := SIN(theta) * q;
  x[0] := ux - a;
  x[1] := ux * Constants.Cos120 - uyi * Constants.Sin120 - a;
  x[2] := ux * Constants.Cos120 + uyi * Constants.Sin120  - a;
  SolveResolvent := 3;
  RETURN;

ELSE
  aa := -cbrt(ABS(rr) + SQRT(r2 - q3));
  IF (rr < 0.0) THEN
    aa := -aa;
  END_IF
  bb := SEL(0.0 = aa, q / aa, 0.0);
  
  x[0] := (aa + bb) - a;
  x[1] := -(aa + bb) / 2 - a;
  x[2] := SQRT(3) * (aa - bb) / 2;
  IF (ABS(x[2]) < Constants.DoubleEpsilon) THEN
    x[2] := x[1];
    SolveResolvent := 2;
    RETURN;
  END_IF
  
  SolveResolvent := 1;
END_IF
END_METHOD

END_PROGRAM

// Struckig/Position/PositionFirstOrderStep1
// Struckig
// Copyright (C) 2022 Stefan Besler

// This program is free software: you can redistribute it and/or modify
// it under the terms of the GNU General Public License as published by
// the Free Software Foundation, either version 3 of the License, or
// (at your option) any later version.

// This program is distributed in the hope that it will be useful,
// but WITHOUT ANY WARRANTY; without even the implied warranty of
// MERCHANTABILITY or FITNESS FOR A PARTICULAR PURPOSE.  See the
// GNU General Public License for more details.
//
// You should have received a copy of the GNU General Public License
// along with THIS PROGRAM.  IF NOT, see <http://www.gnu.org/licenses/>.
/// Mathematical equations for Step 1 in third-order position interface: Extremal profiles
FUNCTION_BLOCK INTERNAL PositionFirstOrderStep1
VAR
  v0 : LREAL;
  vf : LREAL;
  _vMax, _vMin : LREAL;

  // Pre-calculated expressions
  pd : LREAL;  
END_VAR

METHOD Get : BOOL
VAR_INPUT
  input : REFERENCE TO ProfileDesc;
  block : REFERENCE TO Block; 
END_VAR
VAR_INST
  vMax, vMin, aMax, aMin, jMax : LREAL;
  profile : REFERENCE TO ProfileDesc;
END_VAR
profile REF= block.Pmin;
profile.SetBoundary(input);

vf := SEL(pd > 0, _vMin, _vMax);
profile.t[0] := 0;
profile.t[1] := 0;
profile.t[2] := 0;
profile.t[3] := pd / vf;
profile.t[4] := 0;
profile.t[5] := 0;
profile.t[6] := 0;

IF profile.CheckForFirstOrder(ProfileControlSigns.Uddu, ReachedLimits.Vel, vf)
THEN
  block.Tmin := block.Pmin.t_sum[6] + block.Pmin.Brake.Duration + block.Pmin.Accel.Duration;
  Get := TRUE;
END_IF
END_METHOD

METHOD Set
VAR_INPUT
  p0 : LREAL;
  pf : LREAL;
  vMax, vMin : LREAL;
END_VAR
THIS^.v0 := v0;
THIS^.vf := vf;
THIS^._vMax := vMax;
THIS^._vMin := vMin;

pd := pf - p0;
END_METHOD

END_FUNCTION_BLOCK

// Struckig/Profile/ProfileDesc
// Struckig
// Copyright (C) 2022 Stefan Besler

// This program is free software: you can redistribute it and/or modify
// it under the terms of the GNU General Public License as published by
// the Free Software Foundation, either version 3 of the License, or
// (at your option) any later version.

// This program is distributed in the hope that it will be useful,
// but WITHOUT ANY WARRANTY; without even the implied warranty of
// MERCHANTABILITY or FITNESS FOR A PARTICULAR PURPOSE.  See the
// GNU General Public License for more details.
//
// You should have received a copy of the GNU General Public License
// along with THIS PROGRAM.  IF NOT, see <http://www.gnu.org/licenses/>.
/// The state Profile for position, velocity, acceleration and jerk for a single DoF
/// A single-dof kinematic profile with position, velocity, acceleration and jerk
{attribute 'hide'}
FUNCTION_BLOCK ProfileDesc
VAR_INPUT
  Limits : ReachedLimits;
  Direction : ProfileDirection;
  ControlSigns : ProfileControlSigns;
  
  t, t_sum, j : ARRAY[0..6] OF LREAL;
  a, v, p : ARRAY[0..7] OF LREAL;

  pf, vf, af : LREAL; //! Target (final) kinematic state
  Brake, Accel : BrakeProfile; //! Brake sub-profiles
END_VAR

METHOD Bound : ProfileBound
VAR_INPUT
END_VAR
VAR
  i : INT;
  t_current_sum : LREAL;
END_VAR
Bound.Minimum := Constants.Infinity;
Bound.Maximum := -Constants.Infinity;

IF Brake.Duration > 0.0
THEN
  IF (Brake.t[0] > 0.0)
  THEN
    CheckStepForBound(0.0, Brake.t[0], Brake.p[0], Brake.v[0], Brake.a[0], Brake.j[0], Bound);
  
    IF (Brake.t[1] > 0.0) 
    THEN
      CheckStepForBound(Brake.t[0], Brake.t[1], Brake.p[1], Brake.v[1], Brake.a[1], Brake.j[1], Bound);
      
      IF (Brake.t[2] > 0.0)
      THEN
        CheckStepForBound(Brake.t[0] + Brake.t[1], Brake.t[2], Brake.p[2], Brake.v[2], Brake.a[2], Brake.j[2], Bound);
      END_IF
    END_IF
  END_IF
END_IF

t_current_sum := 0;        
FOR i:=0 TO 6
DO
  IF i > 0
  THEN
    t_current_sum := t_sum[i-1];
	END_IF
  
  CheckStepForBound(t_current_sum + Brake.Duration, t[i], p[i], v[i], a[i], j[i], Bound);
END_FOR 

IF (pf < Bound.Minimum)
THEN
  Bound.Minimum := pf;
  Bound.Tmin := t_sum[6] + Brake.Duration;
END_IF 


IF (pf > Bound.Maximum) 
THEN
  Bound.Maximum := pf;
  Bound.Tmax := t_sum[6] + Brake.Duration;
END_IF
END_METHOD

METHOD CheckBound : BOOL
VAR_INPUT
  t_ext, t_sum, t, p, v, a, j : LREAL;
END_VAR
VAR_IN_OUT
  b : ProfileBound;     
END_VAR
VAR
  p_ext, v_Ext, a_ext : LREAL;
END_VAR
IF (0 < t_ext AND_THEN t_ext < t)
THEN
  Integrate(t_ext, p, v, a, j, p:=p_ext, v:=v_ext, a:=a_ext);
  IF (a_ext > 0 AND_THEN p_ext < b.Minimum)
  THEN
    b.Minimum := p_ext;
    b.Tmin := t_sum + t_ext;
   ELSIF (a_ext < 0 AND_THEN p_ext > b.Maximum) 
   THEN
    b.Maximum := p_ext;
    b.Tmax := t_sum + t_ext; 
  END_IF
END_IF
END_METHOD

/// For velocity interface
METHOD CheckForFirstOrder : BOOL
VAR_INPUT
  controlSigns : ProfileControlSigns;
  limits : ReachedLimits;  
  vUp : LREAL;
END_VAR
VAR
  i : INT;
  vUppLim : LREAL;
  vLowLim : LREAL;
  v_a_zero : LREAL;
END_VAR
// ReachedLimits::VEL
IF t[3] < 0.0
THEN
  RETURN;
END_IF

t_sum[0] := 0;
t_sum[1] := 0;
t_sum[2] := 0;
t_sum[3] := t[3];
t_sum[4] := t[3];
t_sum[5] := t[3];
t_sum[6] := t[3];

IF t_sum[6] > Constants.Tmax // For numerical reasons, is that needed?}
THEN
  RETURN;        
END_IF

j[0] := 0;
j[1] := 0;
j[2] := 0;
j[3] := 0;
j[4] := 0;
j[5] := 0;
j[6] := 0;

a[0] := 0;
a[1] := 0;
a[2] := 0;
a[3] := 0;
a[4] := 0;
a[5] := 0;
a[6] := 0;
a[7] := af;

v[0] := 0;
v[1] := 0;
v[2] := 0;
v[3] := SEL(t[3] > 0, 0, vUp);
v[4] := 0;
v[5] := 0;
v[6] := 0;
v[7] := vf;

FOR i:= 0 TO 6 
DO
  p[i+1] := p[i] + t[i] * (v[i] + t[i] * a[i] / 2);
END_FOR

THIS^.Direction := SEL(vUp > 0, ProfileDirection.Down, ProfileDirection.Up);
THIS^.ControlSigns := controlSigns;
THIS^.Limits := limits;

// Velocity limit can be broken in the beginning if both initial velocity and acceleration are too high
CheckForFirstOrder := ABS(p[7] - pf) < Constants.PositionPrecision;
END_METHOD

/// For velocity interface
METHOD CheckForFirstOrderWithTiming : BOOL
VAR_INPUT
  controlSigns : ProfileControlSigns;
  limits : ReachedLimits;  
  vUp : LREAL;
END_VAR
VAR
  i : INT;
  aUppLim : LREAL;
  aLowLim : LREAL;
END_VAR
CheckForFirstOrderWithTiming := CheckForFirstOrder(controlSigns, limits, vUp); // AND_THEN (ABS(t[6] - tf) < t_precision);
END_METHOD

/// For velocity interface
METHOD CheckForFirstOrderWithTiming2 : BOOL
VAR_INPUT
  controlSigns : ProfileControlSigns;
  limits : ReachedLimits;  
  tf : LREAL;
  vUp : LREAL;
  vMax, vMin : LREAL;
END_VAR
CheckForFirstOrderWithTiming2 :=
  (vMin - Constants.VelocityEpsilon < vUp)
  AND_THEN (vUp < vMax + Constants.VelocityEpsilon)
  AND_THEN CheckForFirstOrderWithTiming(controlSigns, limits, vUp);
END_METHOD

/// For velocity interface
METHOD CheckForSecondOrder : BOOL
VAR_INPUT
  controlSigns : ProfileControlSigns;
  limits : ReachedLimits;  
  aUp, aDown : LREAL;
  vMax, vMin : LREAL;
END_VAR
VAR
  i : INT;
  vUppLim : LREAL;
  vLowLim : LREAL;
  v_a_zero : LREAL;
END_VAR
// ReachedLimits::ACC0
IF t[0] < 0.0
THEN
  RETURN;
END_IF

t_sum[0] := t[0];
FOR i:=0 TO 5
DO
  IF (t[i+1] < 0)
  THEN
    RETURN;
  END_IF
  
  t_sum[i+1] := t_sum[i] + t[i+1];  
END_FOR

IF t_sum[6] > Constants.Tmax // For numerical reasons, is that needed?}
THEN
  RETURN;        
END_IF

j[0] := 0;
j[1] := 0;
j[2] := 0;
j[3] := 0;
j[4] := 0;
j[5] := 0;
j[6] := 0;

IF controlSigns = ProfileControlSigns.Uddu
THEN
  a[0] := SEL(t[0] > 0, 0, aUp);
  a[1] := 0;
  a[2] := SEL(t[2] > 0, 0, aDown);
  a[3] := 0;
  a[4] := SEL(t[4] > 0, 0, aDown);
  a[5] := 0;
  a[6] := SEL(t[6] > 0, 0, aUp);
  a[7] := af;
ELSE
  a[0] := SEL(t[0] > 0, 0, aUp);
  a[1] := 0;
  a[2] := SEL(t[2] > 0, 0, aDown);
  a[3] := 0;
  a[4] := SEL(t[4] > 0, 0, aUp);
  a[5] := 0;
  a[6] := SEL(t[6] > 0, 0, aDown);
  a[7] := af;
END_IF

direction := SEL(vMax > 0, ProfileDirection.Down, ProfileDirection.Up);
vUppLim := SEL(direction = ProfileDirection.Up, vMin, vMax) + Constants.VelocityEpsilon;
vLowLim := SEL(direction = ProfileDirection.Up, vMax, vMin) - Constants.VelocityEpsilon;

FOR i:= 0 TO 6 
DO
  v[i+1] := v[i] + t[i] * a[i];
  p[i+1] := p[i] + t[i] * (v[i] + t[i] * a[i] / 2);
END_FOR


THIS^.ControlSigns := controlSigns;
THIS^.Limits := limits;

// Velocity limit can be broken in the beginning if both initial velocity and acceleration are too high
CheckForSecondOrder := ABS(p[7] - pf) < Constants.PositionPrecision AND_THEN ABS(v[7] - vf) < Constants.VelocityPrecision
    AND_THEN v[2] <= vUppLim AND_THEN v[3] <= vUppLim AND_THEN v[4] <= vUppLim AND_THEN v[5] <= vUppLim AND_THEN v[6] <= vUppLim
    AND_THEN v[2] >= vLowLim AND_THEN v[3] >= vLowLim AND_THEN v[4] >= vLowLim AND_THEN v[5] >= vLowLim AND_THEN v[6] >= vLowLim;
END_METHOD

/// For velocity interface
METHOD CheckForSecondOrderVelocity : BOOL
VAR_INPUT
  controlSigns : ProfileControlSigns;
  limits : ReachedLimits;  
  aUp : LREAL;
END_VAR
VAR
  i : INT;
  aUppLim : LREAL;
  aLowLim : LREAL;
END_VAR
// ReachedLimits::ACC0
IF t[1] < 0.0
THEN
  RETURN;
END_IF

t_sum[0] := 0;
t_sum[1] := t[1];
t_sum[2] := t[1];
t_sum[3] := t[1];
t_sum[4] := t[1];
t_sum[5] := t[1];
t_sum[6] := t[1];

// For numerical reasons, is that needed?
IF t_sum[6] > Constants.Tmax
THEN
  RETURN;
END_IF


j[0] := 0;
j[1] := 0;
j[2] := 0;
j[3] := 0;
j[4] := 0;
j[5] := 0;
j[6] := 0;

a[0] := 0;
a[1] := aUp;
a[2] := 0;
a[3] := 0;
a[4] := 0;
a[5] := 0;
a[6] := 0;
a[7] := THIS^.af;

FOR i:=0 TO 6
DO
  v[i+1] := v[i] + t[i] * a[i];
  p[i+1] := p[i] + t[i] * (v[i] + t[i] * a[i] / 2);
END_FOR

THIS^.ControlSigns := controlSigns;
THIS^.Limits := limits;
THIS^.Direction := SEL(aUp > 0, ProfileDirection.Down, ProfileDirection.Up);

// Velocity limit can be broken in the beginning if both initial velocity and acceleration are too high
CheckForSecondOrderVelocity := ABS(v[6] - vf) < Constants.VelocityPrecision;
END_METHOD

/// For velocity interface
METHOD CheckForSecondOrderVelocityWithTiming : BOOL
VAR_INPUT
  controlSigns : ProfileControlSigns;
  limits : ReachedLimits;  
  aUp : LREAL;
END_VAR
CheckForSecondOrderVelocityWithTiming := CheckForSecondOrderVelocity(controlSigns, limits, aUp); // AND_THEN (ABS(t[6] - tf) < t_precision);
END_METHOD

/// For velocity interface
METHOD CheckForSecondOrderVelocityWithTiming2 : BOOL
VAR_INPUT
  controlSigns : ProfileControlSigns;
  limits : ReachedLimits;  
  tf : LREAL;
  aUp : LREAL;
  aMax : LREAL;
  aMin : LREAL;
END_VAR
CheckForSecondOrderVelocityWithTiming2 :=
 (aMin - Constants.AccelerationEpsilon < aUp)
 AND_THEN (aUp < aMax + Constants.AccelerationEpsilon)
 AND_THEN CheckForSecondOrderVelocityWithTiming(controlSigns, limits, aUp); // AND_THEN (ABS(t[6] - tf) < t_precision);
END_METHOD

/// For velocity interface
METHOD CheckForSecondOrderWithTiming : BOOL
VAR_INPUT
  controlSigns : ProfileControlSigns;
  limits : ReachedLimits;  
  tf : LREAL;
  aUp, aDown : LREAL;
  vMax, vMin : LREAL;
END_VAR
CheckForSecondOrderWithTiming := CheckForSecondOrder(controlSigns, limits, aUp, aDown, vMax, vMin);
END_METHOD

/// For velocity interface
METHOD CheckForSecondOrderWithTiming2 : BOOL
VAR_INPUT
  controlSigns : ProfileControlSigns;
  limits : ReachedLimits;  
  tf : LREAL;
  aUp, aDown : LREAL;
  vMax, vMin : LREAL;
  aMax, aMin : LREAL;  
END_VAR
CheckForSecondOrderWithTiming2 := 
    (aMin - Constants.AccelerationEpsilon < aUp)
    AND_THEN (aUp < aMax + Constants.AccelerationEpsilon)
    AND_THEN (aMin - Constants.AccelerationEpsilon < aDown)
    AND_THEN (aDown < aMax + Constants.AccelerationEpsilon)
    AND_THEN CheckForSecondOrderWithTiming(controlSigns, limits,tf, aUp, aDown, vMax, vMin);
END_METHOD

/// For velocity interface
METHOD CheckForVelocity : BOOL
VAR_INPUT
  controlSigns : ProfileControlSigns;
  limits : ReachedLimits;  
  jf : LREAL;
  aMax : LREAL;
  aMin : LREAL;  
END_VAR
VAR
  i : INT;
  aUppLim : LREAL;
  aLowLim : LREAL;
END_VAR
IF (t[0] < 0)
THEN
  RETURN;
END_IF

t_sum[0] := t[0];
FOR i:=0 TO 5
DO
  IF (t[i+1] < 0)
  THEN
    RETURN;
  END_IF
  
  t_sum[i+1] := t_sum[i] + t[i+1];
END_FOR


IF limits = ReachedLimits.Acc0
THEN
  IF t[1] < Constants.DoubleEpsilon
  THEN
    RETURN;
  END_IF
END_IF


IF t_sum[6] > Constants.Tmax // For numerical reasons, is that needed?}
THEN
  RETURN;        
END_IF

IF controlSigns = ProfileControlSigns.Uddu
THEN
  j[0] := SEL(t[0] > 0, 0, jf);
  j[1] := 0;
  j[2] := SEL(t[2] > 0, 0, -jf);
  j[3] := 0;
  j[4] := SEL(t[4] > 0, 0, -jf);
  j[5] := 0;
  j[6] := SEL(t[6] > 0, 0, jf);          
ELSE
  j[0] := SEL(t[0] > 0, 0, jf);
  j[1] := 0;
  j[2] := SEL(t[2] > 0, 0, -jf);
  j[3] := 0;
  j[4] := SEL(t[4] > 0, 0, jf);
  j[5] := 0;
  j[6] := SEL(t[6] > 0, 0, -jf); 
END_IF


FOR i:=0 TO 6
DO
  a[i+1] := a[i] + t[i] * j[i];
  v[i+1] := v[i] + t[i] * (a[i] + t[i] * j[i] / 2);
  p[i+1] := p[i] + t[i] * (v[i] + t[i] * (a[i] / 2 + t[i] * j[i] / 6));        
END_FOR

      
THIS^.ControlSigns := controlSigns;
THIS^.Limits := limits;

aUppLim := SEL((aMax > 0), aMin, aMax) + 5E-12;
aLowLim := SEL((aMax > 0), aMax, aMin) - 5E-12;

// Velocity limit can be broken in the beginning if both initial velocity and acceleration are too high
CheckForVelocity := ABS(v[7] - vf) < Constants.VelocityPrecision
    AND_THEN ABS(a[7] - af) < Constants.AccelerationPrecision // This is not really needed, but we want to double check
    AND_THEN a[1] >= aLowLim AND_THEN a[3] >= aLowLim AND_THEN a[5] >= aLowLim
    AND_THEN a[1] <= aUppLim AND_THEN a[3] <= aUppLim AND_THEN a[5] <= aUppLim;
END_METHOD

/// For velocity interface
METHOD CheckForVelocityWithTiming : BOOL
VAR_INPUT
  controlSigns : ProfileControlSigns;
  limits : ReachedLimits;  
  jf : LREAL;
  aMax : LREAL;
  aMin : LREAL;  
  jMax : LREAL;  
END_VAR
// Time doesn't need to be checked as every profile has a: tf - ... equation
CheckForVelocityWithTiming := (ABS(jf) < ABS(jMax) + Constants.JerkEpsilon) AND_THEN CheckForVelocity(controlSigns, limits, jf, aMax, aMin);
END_METHOD

METHOD CheckStepForBound : BOOL
VAR_INPUT
  t_sum, t, p, v, a, j : LREAL;
END_VAR
VAR_IN_OUT
  b : ProfileBound;  
END_VAR
VAR
  d, d_sqrt : LREAL;
END_VAR
IF (p < b.Minimum)
THEN 
  b.Minimum := p;
  b.Tmin := t_sum;
END_IF

IF (p > b.Maximum)
THEN 
  b.Maximum := p;
  b.Tmax := t_sum;
END_IF

IF (j <> 0) 
THEN
  d := a * a - 2 * j * v;
  IF (ABS(d) < Constants.DoubleEpsilon)
  THEN
    CheckBound(-a / j, t_sum, t, p, v, a, j, b:=b);
   ELSIF (d > 0) 
   THEN
    d_sqrt := SQRT(d);
    CheckBound((-a - D_sqrt) / j, t_sum, t, p, v, a, j, b:=b);
    CheckBound((-a + D_sqrt) / j, t_sum, t, p, v, a, j, b:=b);           
  END_IF
END_IF
END_METHOD

/// For position interface
METHOD CheckVel : BOOL
VAR_INPUT
  controlSigns : ProfileControlSigns;    
  limits : ReachedLimits;
  jf : LREAL;
  vMax : LREAL;
  vMin : LREAL;  
  aMax : LREAL;
  aMin : LREAL;
  setLimits : BOOL;
END_VAR
VAR
  i : INT;
  v_a_zero : LREAL;
  vUppLim, vLowLim : LREAL;  
  aUppLim, aLowLim : LREAL;
END_VAR
IF (t[0] < 0) 
THEN
  RETURN;
END_IF

t_sum[0] := t[0];
FOR i:=0 TO 5
DO
  IF (t[i+1] < 0)
  THEN
    RETURN;
  END_IF
  
  t_sum[i+1] := t_sum[i] + t[i+1];  
END_FOR

IF limits = ReachedLimits.Acc0Acc1Vel OR_ELSE limits = ReachedLimits.Acc0Vel OR_ELSE limits = ReachedLimits.Acc1Vel OR_ELSE limits = ReachedLimits.Vel THEN
  IF (t[3] < Constants.DoubleEpsilon) 
  THEN
    RETURN;                    
  END_IF
END_IF

IF limits = ReachedLimits.Acc0 OR_ELSE limits = ReachedLimits.Acc0Acc1
THEN
  IF (t[1] < Constants.DoubleEpsilon) 
  THEN
    RETURN;                    
  END_IF
END_IF

IF limits = ReachedLimits.Acc1 OR_ELSE limits = ReachedLimits.Acc0Acc1
THEN
  IF (t[5] < Constants.DoubleEpsilon)
  THEN
    RETURN;            
  END_IF
END_IF

IF t_sum[6] > Constants.Tmax  // For numerical reasons, is that needed?
THEN
  RETURN;        
END_IF
        
IF controlSigns = ProfileControlSigns.Uddu
THEN
  j[0] := SEL(t[0] > 0, 0, jf);
  j[1] := 0;
  j[2] := SEL(t[2] > 0, 0, -jf);
  j[3] := 0;
  j[4] := SEL(t[4] > 0, 0, -jf);
  j[5] := 0;
  j[6] := SEL(t[6] > 0, 0, jf);          
ELSE
  j[0] := SEL(t[0] > 0, 0, jf);
  j[1] := 0;
  j[2] := SEL(t[2] > 0, 0, -jf);
  j[3] := 0;
  j[4] := SEL(t[4] > 0, 0, jf);
  j[5] := 0;
  j[6] := SEL(t[6] > 0, 0, -jf); 
END_IF

vUppLim := SEL(vMax > 0, vMin, vMax) + 1E-12;
vLowLim := SEL(vMax > 0, vMax, vMin) - 1E-12;

direction := SEL(vMax > 0, ProfileDirection.Down, ProfileDirection.Up);
vUppLim := SEL(direction = ProfileDirection.Up, vMin, vMax) + Constants.VelocityEpsilon;
vLowLim := SEL(direction = ProfileDirection.Up, vMax, vMin) - Constants.VelocityEpsilon;
        
FOR i:= 0 TO 6 
DO
  a[i+1] := a[i] + t[i] * j[i];
  v[i+1] := v[i] + t[i] * (a[i] + t[i] * j[i] / 2);
  p[i+1] := p[i] + t[i] * (v[i] + t[i] * (a[i] / 2 + t[i] * j[i] / 6));

  IF limits = ReachedLimits.Acc0Acc1Vel OR_ELSE limits = ReachedLimits.Acc0Acc1 OR_ELSE limits = ReachedLimits.Acc0Vel OR_ELSE limits = ReachedLimits.Acc1Vel OR_ELSE limits = ReachedLimits.Vel
  THEN
    IF i = 2
    THEN
     a[3] := 0.0;
    END_IF
  END_IF
  
  IF setLimits
  THEN
    IF limits = ReachedLimits.Acc1
    THEN
      IF i = 2
      THEN
        a[3] := aMin;
      END_IF
    ELSIF limits = ReachedLimits.Acc0Acc1
    THEN
      CASE i
      OF
      0: a[1] := aMax;
      4: a[5] := aMin;
      END_CASE  
    END_IF
  END_IF
  
  IF (i > 1 AND_THEN a[i+1] * a[i] < -Constants.DoubleEpsilon) 
  THEN
    v_a_zero := v[i] - (a[i] * a[i]) / (2 * j[i]);
    IF (v_a_zero > vUppLim OR_ELSE v_a_zero < vLowLim)
    THEN
      RETURN;        
		END_IF
  END_IF
END_FOR


THIS^.ControlSigns := controlSigns;
THIS^.Limits := limits;

aUppLim := SEL(direction = ProfileDirection.Up, aMin, aMax) + Constants.AccelerationEpsilon;
aLowLim := SEL(direction = ProfileDirection.Up, aMax, aMin) - Constants.AccelerationEpsilon;

// Velocity limit can be broken in the beginning if both initial velocity and acceleration are too high
CheckVel := ABS(p[7] - pf) < Constants.PositionPrecision
    AND_THEN ABS(v[7] - vf) < Constants.VelocityPrecision
    AND_THEN ABS(a[7] - af) < Constants.AccelerationPrecision // This is not really needed, but we want to double check
    // AND_THEN ABS(v[3]) <= vMaxAbs AND_THEN ABS(v[4]) <= vMaxAbs AND_THEN ABS(v[5]) <= vMaxAbs AND_THEN ABS(v[6]) <= vMaxAbs
    AND_THEN a[1] >= aLowLim AND_THEN a[3] >= aLowLim AND_THEN a[5] >= aLowLim
    AND_THEN a[1] <= aUppLim AND_THEN a[3] <= aUppLim AND_THEN a[5] <= aUppLim
    AND_THEN v[3] <= vUppLim AND_THEN v[4] <= vUppLim AND_THEN v[5] <= vUppLim AND_THEN v[6] <= vUppLim
    AND_THEN v[3] >= vLowLim AND_THEN v[4] >= vLowLim AND_THEN v[5] >= vLowLim AND_THEN v[6] >= vLowLim; // this is not really needed, but we want to double check
END_METHOD

METHOD CheckWithTiming : BOOL
VAR_INPUT
  controlSigns : ProfileControlSigns;    
  limits : ReachedLimits;
  tf : LREAL;
  jf : LREAL;
  vMax : LREAL;
  vMin : LREAL;  
  aMax : LREAL;
  aMin : LREAL;  
END_VAR
// Time doesn't need to be checked as every Profile has a: tf - ... equation
CheckWithTiming := CheckVel(controlSigns, limits, jf, vMax, vMin, aMax, aMin, setLimits:=FALSE); // && (std::abs(t_sum[6] - tf) < Constants.TimePrecision)
END_METHOD

METHOD CheckWithTiming2 : BOOL
VAR_INPUT
  controlSigns : ProfileControlSigns;    
  limits : ReachedLimits;
  tf : LREAL;
  jf : LREAL;
  vMax : LREAL;
  vMin : LREAL;  
  aMax : LREAL;
  aMin : LREAL;
  jMax  : LREAL;
END_VAR
CheckWithTiming2 := (ABS(jf) < ABS(jMax) + Constants.JerkEpsilon) AND_THEN CheckWithTiming(controlSigns, limits, tf, jf, vMax, vMin, aMax, aMin);
END_METHOD

METHOD FirstStateAtPosition : BOOL
VAR_INPUT
  pt, offset : LREAL;
END_VAR
VAR_IN_OUT
  t_t, v_t, a_t : LREAL;
END_VAR
VAR
  i,h : INT;
  p_t : LREAL;
  polynom : ARRAY[0..4] OF LREAL;
  rootCount : INT;
  root : ARRAY[0..6] OF LREAL;
END_VAR
FOR i:=0 TO 6
DO
  IF ABS(p[i] - pt) < Constants.DoubleEpsilon
  THEN
    t_t := offset + SEL(i>0, 0, t_sum[i-1]);
    v_t := v[i];
    a_t := a[i];
    FirstStateAtPosition := TRUE;
    RETURN;
	END_IF
  
  IF t[i] = 0
  THEN
    CONTINUE;
	END_IF
  
  polynom[0] := j[i]/6;
  polynom[1] := a[i]*0.5;
  polynom[2] := v[i];
  polynom[3] := p[i]-pt;
  Roots.SolveCub(ADR(polynom), rootCount:=rootCount, roots:=root);
  FOR h:=0 TO rootCount
  DO
    IF(0 < root[h] AND_THEN root[h] <= t[i])
    THEN
      t_t := offset + root[h] + SEL(i>0, 0, t_sum[i-1]);
      Integrate(root[h], p[i], v[i], a[i], j[i], p_t, v_t, a_t);
      FirstStateAtPosition := TRUE;
      RETURN;      
		END_IF
  END_FOR
  
END_FOR

IF ABS(pf-pt) < Constants.Epsilon
THEN
  t_t := offset + t_sum[6];
  v_t := vf;
  a_t := af;
  FirstStateAtPosition := TRUE;
  RETURN;      
END_IF
END_METHOD

/// Set boundary values for the position interface
METHOD SetBoundary
VAR_IN_OUT CONSTANT
  profile : ProfileDesc;
END_VAR
a[0] := profile.a[0];
v[0] := profile.v[0];
p[0] := profile.p[0];
af := profile.af;
vf := profile.vf;
pf := profile.pf;
Brake := profile.Brake;
Accel := profile.Accel;
END_METHOD

/// Set boundary values for the position interface
METHOD SetBoundaryPosition
VAR_INPUT
  p0_new, v0_new, a0_new, pf_new, vf_new, af_new : LREAL;
END_VAR
a[0] := a0_new;
v[0] := v0_new;
p[0] := p0_new;
af := af_new;
vf := vf_new;
pf := pf_new;
END_METHOD

/// Set boundary values for the velocity interface
METHOD SetBoundaryVelocity
VAR_INPUT
  p0_new, v0_new, a0_new, vf_new, af_new : LREAL;
END_VAR
a[0] := a0_new;
v[0] := v0_new;
p[0] := p0_new;
af := af_new;
vf := vf_new;
END_METHOD

END_FUNCTION_BLOCK

// Struckig/Position/PositionFirstOrderStep2
// Struckig
// Copyright (C) 2022 Stefan Besler

// This program is free software: you can redistribute it and/or modify
// it under the terms of the GNU General Public License as published by
// the Free Software Foundation, either version 3 of the License, or
// (at your option) any later version.

// This program is distributed in the hope that it will be useful,
// but WITHOUT ANY WARRANTY; without even the implied warranty of
// MERCHANTABILITY or FITNESS FOR A PARTICULAR PURPOSE.  See the
// GNU General Public License for more details.
//
// You should have received a copy of the GNU General Public License
// along with THIS PROGRAM.  IF NOT, see <http://www.gnu.org/licenses/>.
/// Mathematical equations for Step 2 in third-order position interface: Time synchronization
FUNCTION_BLOCK INTERNAL PositionFirstOrderStep2
VAR
  minimize_jerk : BOOL;
  v0, a0 : LREAL;
  tf, vf, af : LREAL;
  _vMax, _vMin : LREAL;
  
  // Pre-calculated expressions
  pd : LREAL;
  tf_tf, tf_p3, tf_p4 : LREAL;
  vd, vd_vd : LREAL;
  ad, ad_ad : LREAL;
  v0_v0, vf_vf : LREAL;
  a0_a0, a0_p3, a0_p4, a0_p5, a0_p6 : LREAL;
  af_af, af_p3, af_p4, af_p5, af_p6 : LREAL;
  jMax_jMax : LREAL;
  g1, g2 : LREAL;
  t_min, t_max : LREAL;
  up_first : BOOL;
  
  d_extremasCount : INT;
  d_extremas : ARRAY[0..6] OF LREAL;
  indices : ARRAY[0..6] OF INT;
  
  h0, h0a, h0b, h0c, h1, h2 : LREAL;  
  h3, jf : LREAL;  
  ph1, ph2, ph3, ph4 : LREAL;
  t : LREAL; 
  orig, deriv : LREAL;
  i : INT;
  ph0, ph5, ph6, ph7 : LREAL;
  h1a : LREAL;
  p1, val_max : LREAL;
  polynom, deriva, dderiv, ddderiv, root : ARRAY[0..6] OF LREAL;
  dd_tz_intervals : ARRAY[0..6, 0..1] OF LREAL;
  tz, tz_max, tz_current, dd_tz_current, tz_min : LREAL; 
  deriv_newton, res, p_val, val_new : LREAL;    
END_VAR

METHOD Get : BOOL
VAR_INPUT
  profile : REFERENCE TO ProfileDesc;
END_VAR
vf := pd / tf;

profile.t[0] := 0;
profile.t[1] := 0;
profile.t[2] := 0;
profile.t[3] := tf;
profile.t[4] := 0;
profile.t[5] := 0;
profile.t[6] := 0;

Get := profile.CheckForFirstOrderWithTiming2(ProfileControlSigns.Uddu, ReachedLimits.None, tf, vf, _vMax, _vMin);
END_METHOD

METHOD Set
VAR_INPUT
  tf : LREAL;
  p0 : LREAL;
  pf : LREAL;
  vMax, vMin : LREAL;
END_VAR
THIS^.tf := tf;
THIS^.v0 := v0;
THIS^.vf := vf;
THIS^._vMax := vMax;
THIS^._vMin := vMin;

pd := pf - p0;
vd := vf - v0;
END_METHOD

END_FUNCTION_BLOCK

// Struckig/Position/PositionSecondOrderStep1
// Struckig
// Copyright (C) 2022 Stefan Besler

// This program is free software: you can redistribute it and/or modify
// it under the terms of the GNU General Public License as published by
// the Free Software Foundation, either version 3 of the License, or
// (at your option) any later version.

// This program is distributed in the hope that it will be useful,
// but WITHOUT ANY WARRANTY; without even the implied warranty of
// MERCHANTABILITY or FITNESS FOR A PARTICULAR PURPOSE.  See the
// GNU General Public License for more details.
//
// You should have received a copy of the GNU General Public License
// along with THIS PROGRAM.  IF NOT, see <http://www.gnu.org/licenses/>.
/// Mathematical equations for Step 1 in third-order position interface: Extremal profiles
FUNCTION_BLOCK INTERNAL PositionSecondOrderStep1
VAR
  v0 : LREAL;
  vf : LREAL;
  _vMax, _vMin, _aMax, _aMin : LREAL;

  // Pre-calculated expressions
  pd : LREAL;
  h1 : LREAL;
  
  validProfiles : ARRAY[0..5] OF ProfileDesc; // Max 5 valid profiles + 1 spare for numerical issues
  validProfileCounter : INT := -1;
  
  left_duration, right_duration : LREAL;    
END_VAR

METHOD AddInterval
VAR_IN_OUT
  interval : BlockInterval;
  Left : ProfileDesc;
  Right : ProfileDesc;
END_VAR
left_duration := Left.t_sum[6] + Left.Brake.Duration + Left.Accel.Duration;
right_duration := Right.t_sum[6] + Right.Brake.Duration + Right.Accel.Duration;
IF (left_duration < right_duration)
THEN
  interval.Left := left_duration;
  interval.Right := right_duration;
  interval.Profile := Right;
  interval.IsUsed := TRUE;
ELSE
  interval.Left := right_duration;
  interval.Right := left_duration;
  interval.Profile := Left;
  interval.IsUsed := TRUE;  
END_IF
END_METHOD

METHOD AddProfile
VAR_IN_OUT CONSTANT
  Profile : ProfileDesc;
END_VAR
validProfileCounter := validProfileCounter + 1;
validProfiles[validProfileCounter] := Profile;
END_METHOD

METHOD CalculateBlock : BOOL
VAR_IN_OUT
  block : Block;
END_VAR
VAR
  i, j : INT;
  Tmin : LREAL;
  idx_min : INT;
  idx_else_1, idx_else_2, idx_else_3, idx_else_4 : INT;
END_VAR
block.A.IsUsed := FALSE;
block.B.IsUsed := FALSE;

IF validProfileCounter = 0
THEN
  block.Pmin := validProfiles[0];
  block.Tmin := block.Pmin.t_sum[6] + block.Pmin.Brake.Duration + block.Pmin.Accel.Duration; 
  CalculateBlock := TRUE;

ELSIF validProfileCounter = 1 
THEN

  IF ABS(validProfiles[0].t_sum[6] - validProfiles[1].t_sum[6]) < 8*Constants.Epsilon
  THEN
    block.Pmin := validProfiles[0];
    block.Tmin := block.Pmin.t_sum[6] + block.Pmin.Brake.Duration + block.Pmin.Accel.Duration;  
    CalculateBlock := TRUE;
    RETURN;
	END_IF
  
  IF ParameterList.NumericalRobust
  THEN
    idx_min := SEL(validProfiles[0].t_sum[6] < validProfiles[1].t_sum[6], 1, 0);
    idx_else_1 := (idx_min + 1) MOD 2;

    block.Pmin := validProfiles[idx_min];
    block.Tmin := block.Pmin.t_sum[6] + block.Pmin.Brake.Duration + block.Pmin.Accel.Duration; 
    AddInterval(block.A, validProfiles[idx_min], validProfiles[idx_else_1]);
    CalculateBlock := TRUE;
    RETURN; 
	END_IF

// Only happens due to numerical issues
ELSIF (validProfileCounter = 3) 
THEN
  // Find "identical" profiles
  IF (ABS(validProfiles[0].t_sum[6] - validProfiles[1].t_sum[6]) < 32*Constants.Epsilon AND_THEN validProfiles[0].Direction <> validProfiles[1].Direction)
  THEN
    RemoveProfile(1);
  ELSIF (ABS(validProfiles[2].t_sum[6] - validProfiles[3].t_sum[6]) < 256*Constants.Epsilon  AND_THEN validProfiles[2].Direction <> validProfiles[3].Direction)
  THEN
    RemoveProfile(3);
  ELSIF (ABS(validProfiles[0].t_sum[6] - validProfiles[3].t_sum[6]) < 256*Constants.Epsilon AND_THEN validProfiles[0].Direction <> validProfiles[3].Direction)
  THEN
    RemoveProfile(3);
  ELSE
    RETURN;
  END_IF

ELSIF ((validProfileCounter+1) MOD 2 = 0)
THEN
  RETURN;
END_IF

// Find index of fastest Profile
Tmin := Constants.Infinity;
FOR i:=0 TO validProfileCounter
DO
  FOR j:=0 TO validProfileCounter
  DO
    IF validProfiles[i].t_sum[6] + validProfiles[i].Brake.Duration < validProfiles[j].t_sum[6] + validProfiles[j].Brake.Duration AND_THEN
       validProfiles[i].t_sum[6] + validProfiles[i].Brake.Duration < Tmin
    THEN
      Tmin := validProfiles[i].t_sum[6] + validProfiles[i].Brake.Duration + validProfiles[i].Accel.Duration;
      idx_min := i;
		END_IF
  END_FOR
END_FOR

block.Pmin := validProfiles[idx_min];
block.Tmin := block.Pmin.t_sum[6] + block.Pmin.Brake.Duration + block.Pmin.Accel.Duration;
IF (validProfileCounter = 2)
THEN
  idx_else_1 := (idx_min + 1) MOD 3;
  idx_else_2 := (idx_min + 2) MOD 3;
  
  AddInterval(block.A, validProfiles[idx_else_1], validProfiles[idx_else_2]);
  CalculateBlock := TRUE;
  RETURN;

 ELSIF (validProfileCounter = 4)
 THEN
  idx_else_1 := (idx_min + 1) MOD 5;
  idx_else_2 := (idx_min + 2) MOD 5;
  idx_else_3 := (idx_min + 3) MOD 5;
  idx_else_4 := (idx_min + 4) MOD 5;
  
  IF (validProfiles[idx_else_1].Direction = validProfiles[idx_else_2].Direction)
  THEN
    AddInterval(block.A, validProfiles[idx_else_1], validProfiles[idx_else_2]);
    AddInterval(block.B, validProfiles[idx_else_3], validProfiles[idx_else_4]);
  ELSE 
    AddInterval(block.A, validProfiles[idx_else_1], validProfiles[idx_else_4]);
    AddInterval(block.B, validProfiles[idx_else_2], validProfiles[idx_else_3]);
  END_IF
  
  CalculateBlock := TRUE;
END_IF
END_METHOD

METHOD Get : BOOL
VAR_INPUT
  input : REFERENCE TO ProfileDesc;
  block : REFERENCE TO Block; 
END_VAR
VAR_INST
  vMax, vMin, aMax, aMin, jMax : LREAL;
  profile : REFERENCE TO ProfileDesc;
END_VAR
validProfileCounter := -1;

// Zero-limits special case
IF _vMax = 0.0 AND_THEN _vMin = 0.0
THEN
  block.Pmin.SetBoundary(input);

  IF time_all_single_step(block.Pmin, _vMax, _vMin, _aMax, _aMin) 
  THEN
    block.Tmin := block.Pmin.t_sum[6] + block.Pmin.Brake.Duration + block.Pmin.Accel.Duration;
    AddInterval(block.A, block.Pmin, block.Pmin);
    
    IF ABS(v0) > Constants.DoubleEpsilon 
    THEN
	    block.A.Left := block.Tmin;
      block.A.Right := Constants.Infinity;
    END_IF
    
    Get := TRUE;
    RETURN; 
  END_IF
  
  RETURN;
END_IF

validProfiles[0].SetBoundary(input);

IF ABS(vf) < Constants.DoubleEpsilon
THEN
  // There is no blocked interval when vf==0, so return after first found profile
  vMax := SEL(pd >= 0, _vMin, _vMax);
  vMin := SEL(pd >= 0, _vMax, _vMin);
  aMax := SEL(pd >= 0, _aMin, _aMax);
  aMin := SEL(pd >= 0, _aMax, _aMin);
  
  time_none(input, vMax, vMin, aMax, aMin, TRUE);
  IF (validProfileCounter >= 0) THEN
    Get := CalculateBlock(block);
    RETURN;
  END_IF
  
  time_acc0(input, vMax, vMin, aMax, aMin, TRUE);
  IF (validProfileCounter >= 0) THEN
    Get := CalculateBlock(block);
    RETURN;
  END_IF
  
  time_none(input, vMin, vMax, aMin, aMax, TRUE);
  IF (validProfileCounter >= 0) THEN
    Get := CalculateBlock(block);
    RETURN;
  END_IF
  
  time_acc0(input, vMin, vMax, aMin, aMax, TRUE);
  IF (validProfileCounter >= 0) THEN
    Get := CalculateBlock(block);
    RETURN;
  END_IF 
ELSE
  time_none(input, _vMax, _vMin, _aMax, _aMin, FALSE);
  time_none(input, _vMin, _vMax, _aMin, _aMax, FALSE);
  time_acc0(input, _vMax, _vMin, _aMax, _aMin, FALSE);
  time_acc0(input, _vMin, _vMax, _aMin, _aMax, FALSE);
  
  IF (validProfileCounter >= 0) THEN
    Get := CalculateBlock(block);
    RETURN;
  END_IF   
END_IF
END_METHOD

METHOD PRIVATE RemoveProfile : BOOL
VAR_INPUT
  index : INT;
END_VAR
VAR
  i : INT;
END_VAR
// todo, this is pretty slow in twincat
FOR i:=index TO validProfileCounter-2
DO
  validProfiles[i] := validProfiles[i + 1];
END_FOR

validProfileCounter := validProfileCounter - 1;
END_METHOD

METHOD Set
VAR_INPUT
  p0, v0 : LREAL;
  pf, vf : LREAL;
  vMax, vMin : LREAL;
  aMax, aMin : LREAL;
END_VAR
THIS^.v0 := v0;
THIS^.vf := vf;
THIS^._vMax := vMax;
THIS^._vMin := vMin;
THIS^._aMax := aMax;
THIS^._aMin := aMin;

pd := pf - p0;
END_METHOD

METHOD PRIVATE time_acc0
VAR_INPUT
  profile : REFERENCE TO ProfileDesc;
  vMax, vMin, aMax, aMin : LREAL;
  return_after_found : BOOL;  
END_VAR
profile.t[0] := (-v0 + vMax)/aMax;
profile.t[1] :=(aMin*v0*v0 - aMax*vf*vf)/(2*aMax*aMin*vMax) + vMax*(aMax - aMin)/(2*aMax*aMin) + pd/vMax;
profile.t[2] := (vf - vMax)/aMin;
profile.t[3] := 0;
profile.t[4] := 0;
profile.t[5] := 0;
profile.t[6] := 0;

IF profile.CheckForSecondOrder(ProfileControlSigns.Uddu, ReachedLimits.Acc0, aMax, aMin, vMax, vMin)
THEN
  AddProfile(profile);
END_IF
END_METHOD

METHOD PRIVATE time_all_single_step : BOOL
VAR_INPUT
  profile : REFERENCE TO ProfileDesc;
  vMax, vMin, aMax, aMin : LREAL;
END_VAR
IF ABS(vf - v0) > Constants.DoubleEpsilon
THEN
  RETURN;
END_IF

profile.t[0] := 0;
profile.t[1] := 0;
profile.t[2] := 0;
profile.t[3] := 0;
profile.t[4] := 0;
profile.t[5] := 0;
profile.t[6] := 0;

IF ABS(v0) > Constants.DoubleEpsilon
THEN
  profile.t[3] := pd / v0;
  IF (profile.CheckForSecondOrder(ProfileControlSigns.Uddu, ReachedLimits.None, 0.0, 0.0, vMax, vMin))
  THEN
    time_all_single_step := TRUE;
  END_IF
ELSIF ABS(pd) < Constants.DoubleEpsilon
THEN
  IF (profile.CheckForSecondOrder(ProfileControlSigns.Uddu, ReachedLimits.None, 0.0, 0.0, vMax, vMin))
  THEN
    time_all_single_step := TRUE;
  END_IF
END_IF
END_METHOD

/// Only for numerical issues, always return_after_found
METHOD PRIVATE time_none
VAR_INPUT
  profile : REFERENCE TO ProfileDesc;
  vMax, vMin, aMax, aMin : LREAL;
  return_after_found : BOOL;
END_VAR
h1 := (aMax*vf*vf - aMin*v0*v0 - 2*aMax*aMin*pd)/(aMax - aMin);
IF h1 >= 0.0
THEN
  h1 := SQRT(h1);
  
  // Solution 1
  profile.t[0] := -(v0 + h1)/aMax;
  profile.t[1] := 0;
  profile.t[2] := (vf + h1)/aMin;
  profile.t[3] := 0;
  profile.t[4] := 0;
  profile.t[5] := 0;
  profile.t[6] := 0;  
  IF profile.CheckForSecondOrder(ProfileControlSigns.Uddu, ReachedLimits.None, aMax, aMin, vMax, vMin)
  THEN
    AddProfile(profile);
    IF return_after_found
    THEN
      RETURN;
    END_IF
  END_IF

  
  // Solution 2
  profile.t[0] := (-v0 + h1)/aMax;
  profile.t[1] := 0;
  profile.t[2] := (vf - h1)/aMin;
  profile.t[3] := 0;
  profile.t[4] := 0;
  profile.t[5] := 0;
  profile.t[6] := 0;  
  IF profile.CheckForSecondOrder(ProfileControlSigns.Uddu, ReachedLimits.None, aMax, aMin, vMax, vMin)
  THEN
    AddProfile(profile);
    IF return_after_found
    THEN
      RETURN;
    END_IF
  END_IF
END_IF
END_METHOD

END_FUNCTION_BLOCK

// Struckig/Position/PositionSecondOrderStep2
// Struckig
// Copyright (C) 2022 Stefan Besler

// This program is free software: you can redistribute it and/or modify
// it under the terms of the GNU General Public License as published by
// the Free Software Foundation, either version 3 of the License, or
// (at your option) any later version.

// This program is distributed in the hope that it will be useful,
// but WITHOUT ANY WARRANTY; without even the implied warranty of
// MERCHANTABILITY or FITNESS FOR A PARTICULAR PURPOSE.  See the
// GNU General Public License for more details.
//
// You should have received a copy of the GNU General Public License
// along with THIS PROGRAM.  IF NOT, see <http://www.gnu.org/licenses/>.
/// Mathematical equations for Step 2 in third-order position interface: Time synchronization
FUNCTION_BLOCK INTERNAL PositionSecondOrderStep2
VAR
  minimize_jerk : BOOL;
  v0, a0 : LREAL;
  tf, vf, af : LREAL;
  _vMax, _vMin, _aMax, _aMin : LREAL;
  
  // Pre-calculated expressions
  pd : LREAL;
  tf_tf, tf_p3, tf_p4 : LREAL;
  vd, vd_vd : LREAL;
  ad, ad_ad : LREAL;
  v0_v0, vf_vf : LREAL;
  a0_a0, a0_p3, a0_p4, a0_p5, a0_p6 : LREAL;
  af_af, af_p3, af_p4, af_p5, af_p6 : LREAL;
  jMax_jMax : LREAL;
  g1, g2 : LREAL;
  t_min, t_max : LREAL;
  up_first : BOOL;
  
  d_extremasCount : INT;
  d_extremas : ARRAY[0..6] OF LREAL;
  indices : ARRAY[0..6] OF INT;
  
  h0, h0a, h0b, h0c, h1, h2 : LREAL;  
  h3, jf : LREAL;  
  ph1, ph2, ph3, ph4 : LREAL;
  t : LREAL; 
  orig, deriv : LREAL;
  i : INT;
  ph0, ph5, ph6, ph7 : LREAL;
  h1a : LREAL;
  p1, val_max : LREAL;
  polynom, deriva, dderiv, ddderiv, root : ARRAY[0..6] OF LREAL;
  dd_tz_intervals : ARRAY[0..6, 0..1] OF LREAL;
  tz, tz_max, tz_current, dd_tz_current, tz_min : LREAL; 
  deriv_newton, res, p_val, val_new : LREAL;    
END_VAR

METHOD CheckAll : BOOL
VAR_INPUT
  profile : REFERENCE TO ProfileDesc;
  vMax, vMin, aMax, aMin : LREAL;  
END_VAR
CheckAll := time_acc0(profile, vMax, vMin, aMax, aMin) OR_ELSE
            time_none(profile, vMax, vMin, aMax, aMin);
END_METHOD

METHOD Get : BOOL
VAR_INPUT
  Profile : REFERENCE TO ProfileDesc;
END_VAR
// Test all cases to get ones that match
// However we should guess which one is correct and try them first...
IF pd > 0
THEN
  Get := CheckAll(profile, _vMax, _vMin, _aMax, _aMin) OR_ELSE CheckAll(profile, _vMin, _vMax, _aMin, _aMax);
  RETURN;
END_IF

Get := CheckAll(profile, _vMin, _vMax, _aMin, _aMax) OR_ELSE CheckAll(profile, _vMax, _vMin, _aMax, _aMin);
END_METHOD

METHOD Set
VAR_INPUT
  tf : LREAL;
  p0, v0 : LREAL;
  pf, vf : LREAL;
  vMax, vMin : LREAL;
  aMax, aMin : LREAL;
END_VAR
THIS^.tf := tf;
THIS^.v0 := v0;
THIS^.vf := vf;
THIS^._vMax := vMax;
THIS^._vMin := vMin;
THIS^._aMax := aMax;
THIS^._aMin := aMin;

pd := pf - p0;
vd := vf - v0;
END_METHOD

METHOD PRIVATE time_acc0 : BOOL
VAR_INPUT
  profile : REFERENCE TO ProfileDesc;
  vMax, vMin, aMax, aMin : LREAL;
END_VAR
h1 := (2*aMax*(pd - tf*vf) - 2*aMin*(pd - tf*v0) + vd*vd)/(aMax*aMin) + tf*tf;
IF h1 >= 0
THEN
  h1 := SQRT(h1);

  profile.t[0] := (aMax*vd - aMax*aMin*(tf - h1))/(aMax*(aMax - aMin));
  profile.t[1] := h1;
  profile.t[2] := tf - (profile.t[0] + h1);
  profile.t[3] := 0;
  profile.t[4] := 0;
  profile.t[5] := 0;
  profile.t[6] := 0;

  IF profile.CheckForSecondOrderWithTiming(ProfileControlSigns.Uddu, ReachedLimits.Acc0, tf, aMax, aMin, vMax, vMin)
  THEN
    profile.pf := profile.p[7];
    time_acc0 := TRUE;
    RETURN;
  END_IF
END_IF


// UU Solution
h1 := (-vd + aMax*tf);
IF ABS(h1) > Constants.Epsilon AND_THEN ABS(2*aMax*h1) > Constants.Epsilon
THEN

  profile.t[0] := -vd*vd/(2*aMax*h1) + (pd - v0*tf)/h1;
  profile.t[1] := -vd/aMax + tf;
  profile.t[2] := 0;
  profile.t[3] := 0;
  profile.t[4] := 0;
  profile.t[5] := 0;
  profile.t[6] := tf - (profile.t[0] + profile.t[1]);
  
  IF profile.CheckForSecondOrderWithTiming(ProfileControlSigns.Uddu, ReachedLimits.Acc0, tf, aMax, aMin, vMax, vMin)
  THEN
    profile.pf := profile.p[7];
    time_acc0 := TRUE;
    RETURN;
  END_IF
END_IF


// UU Solution - 2 step
profile.t[0] := 0;
profile.t[1] := -vd/aMax + tf;
profile.t[2] := 0;
profile.t[3] := 0;
profile.t[4] := 0;
profile.t[5] := 0;
profile.t[6] := vd/aMax;

IF profile.CheckForSecondOrderWithTiming(ProfileControlSigns.Uddu, ReachedLimits.Acc0, tf, aMax, aMin, vMax, vMin)
THEN
  profile.pf := profile.p[7];
  time_acc0 := TRUE;
  RETURN;
END_IF
END_METHOD

/// Only for numerical issues, always return_after_found
METHOD PRIVATE time_none : BOOL
VAR_INPUT
  profile : REFERENCE TO ProfileDesc;
  vMax, vMin, aMax, aMin : LREAL;
END_VAR
IF ABS(v0) < Constants.DoubleEpsilon AND_THEN ABS(vf) < Constants.DoubleEpsilon AND_THEN ABS(pd) < Constants.DoubleEpsilon
THEN
  profile.t[0] := 0;
  profile.t[1] := tf;
  profile.t[2] := 0;
  profile.t[3] := 0;
  profile.t[4] := 0;
  profile.t[5] := 0;
  profile.t[6] := 0;

  IF profile.CheckForSecondOrderWithTiming(ProfileControlSigns.Uddu, ReachedLimits.None, tf, aMax, aMin, vMax, vMin)
  THEN
    profile.pf := profile.p[7];
    time_none := TRUE;
    RETURN;        
  END_IF
END_IF

// UD Solution 1/2
h1 := 2*(vf*tf - pd);

IF ABS(vd) > Constants.DoubleEpsilon AND_THEN ABS(h1) > Constants.Epsilon
THEN
  profile.t[0] := h1/vd;
  profile.t[1] := tf - profile.t[0];
  profile.t[2] := 0;
  profile.t[3] := 0;
  profile.t[4] := 0;
  profile.t[5] := 0;
  profile.t[6] := 0;

  af := vd*vd/h1;

  IF ((aMin - 1E-12 < af) AND_THEN (af < aMax + 1E-12) AND_THEN profile.CheckForSecondOrderWithTiming(ProfileControlSigns.Uddu, ReachedLimits.None, tf, af, -af, vMax, vMin))
  THEN
    profile.pf := profile.p[7];
    time_none := TRUE;
    RETURN;        
  END_IF
END_IF
END_METHOD

END_FUNCTION_BLOCK

// Struckig/Position/PositionThirdOrderStep1
// Struckig
// Copyright (C) 2022 Stefan Besler

// This program is free software: you can redistribute it and/or modify
// it under the terms of the GNU General Public License as published by
// the Free Software Foundation, either version 3 of the License, or
// (at your option) any later version.

// This program is distributed in the hope that it will be useful,
// but WITHOUT ANY WARRANTY; without even the implied warranty of
// MERCHANTABILITY or FITNESS FOR A PARTICULAR PURPOSE.  See the
// GNU General Public License for more details.
//
// You should have received a copy of the GNU General Public License
// along with THIS PROGRAM.  IF NOT, see <http://www.gnu.org/licenses/>.
/// Mathematical equations for Step 1 in third-order position interface: Extremal profiles
FUNCTION_BLOCK INTERNAL PositionThirdOrderStep1
VAR
  v0, a0 : LREAL;
  vf, af : LREAL;
  _vMax, _vMin, _aMax, _aMin, _jMax : LREAL;

  // Pre-calculated expressions
  pd : LREAL;
  v0_v0, vf_vf : LREAL;
  a0_a0, a0_p3, a0_p4 : LREAL;
  af_af, af_p3, af_p4 : LREAL;
  jMax_jMax : LREAL;
  
  // runtime  calculated expressions
  polynom_none, polynom_acc0, polynom_acc1 : ARRAY[0..4] OF LREAL;
  orig : LREAL;
  deriv : LREAL;
  t : LREAL;
  i : INT;
  h0, h1, h2, h2_h2, h3, h5, h2_none, h3_acc0, h3_acc1, h0_acc0, h2_acc0, h0_acc1, h2_acc1, q : LREAL;
  t_min, t_max, t_min_none, t_max_none, t_min_acc0, t_max_acc0, t_min_acc1, t_max_acc1 : LREAL;
  t_acc1, t_acc0 : LREAL;
  validProfiles : ARRAY[0..5] OF ProfileDesc; // Max 5 valid profiles + 1 spare for numerical issues
  validProfileCounter : INT := -1;
  
  num_roots_none, num_roots_acc0, num_roots_acc1  : INT;
  roots_none, roots_acc0, roots_acc1 : ARRAY[0..6] OF LREAL;
  roots_none_indices, roots_acc0_indices, roots_acc1_indices : ARRAY[0..6] OF INT;
  left_duration, right_duration : LREAL;   
END_VAR

METHOD AddInterval
VAR_IN_OUT
  interval : BlockInterval;
  Left : ProfileDesc;
  Right : ProfileDesc;
END_VAR
left_duration := Left.t_sum[6] + Left.Brake.Duration + Left.Accel.Duration;
right_duration := Right.t_sum[6] + Right.Brake.Duration + Right.Accel.Duration;
IF (left_duration < right_duration)
THEN
  interval.Left := left_duration;
  interval.Right := right_duration;
  interval.Profile := Right;
  interval.IsUsed := TRUE;
ELSE
  interval.Left := right_duration;
  interval.Right := left_duration;
  interval.Profile := Left;
  interval.IsUsed := TRUE;  
END_IF
END_METHOD

METHOD AddProfile
VAR_IN_OUT CONSTANT
  Profile : ProfileDesc;
END_VAR
validProfileCounter := validProfileCounter + 1;
validProfiles[validProfileCounter] := Profile;
END_METHOD

METHOD CalculateBlock : BOOL
VAR_IN_OUT
  block : Block;
END_VAR
VAR
  i, j : INT;
  Tmin : LREAL;
  idx_min : INT;
  idx_else_1, idx_else_2, idx_else_3, idx_else_4 : INT;
END_VAR
block.A.IsUsed := FALSE;
block.B.IsUsed := FALSE;

IF validProfileCounter = 0
THEN
  block.Pmin := validProfiles[0];
  block.Tmin := block.Pmin.t_sum[6] + block.Pmin.Brake.Duration + block.Pmin.Accel.Duration; 
  CalculateBlock := TRUE;

ELSIF validProfileCounter = 1 
THEN

  IF ABS(validProfiles[0].t_sum[6] - validProfiles[1].t_sum[6]) < 8*Constants.Epsilon
  THEN
    block.Pmin := validProfiles[0];
    block.Tmin := block.Pmin.t_sum[6] + block.Pmin.Brake.Duration + block.Pmin.Accel.Duration;  
    CalculateBlock := TRUE;
    RETURN;
	END_IF
  
  IF ParameterList.NumericalRobust
  THEN
    idx_min := SEL(validProfiles[0].t_sum[6] < validProfiles[1].t_sum[6], 1, 0);
    idx_else_1 := (idx_min + 1) MOD 2;

    block.Pmin := validProfiles[idx_min];
    block.Tmin := block.Pmin.t_sum[6] + block.Pmin.Brake.Duration + block.Pmin.Accel.Duration; 
    AddInterval(block.A, validProfiles[idx_min], validProfiles[idx_else_1]);
    CalculateBlock := TRUE;
    RETURN; 
	END_IF

// Only happens due to numerical issues
ELSIF (validProfileCounter = 3) 
THEN
  // Find "identical" profiles
  IF (ABS(validProfiles[0].t_sum[6] - validProfiles[1].t_sum[6]) < 32*Constants.Epsilon AND_THEN validProfiles[0].Direction <> validProfiles[1].Direction)
  THEN
    RemoveProfile(1);
  ELSIF (ABS(validProfiles[2].t_sum[6] - validProfiles[3].t_sum[6]) < 256*Constants.Epsilon  AND_THEN validProfiles[2].Direction <> validProfiles[3].Direction)
  THEN
    RemoveProfile(3);
  ELSIF (ABS(validProfiles[0].t_sum[6] - validProfiles[3].t_sum[6]) < 256*Constants.Epsilon AND_THEN validProfiles[0].Direction <> validProfiles[3].Direction)
  THEN
    RemoveProfile(3);
  ELSE
    RETURN;
  END_IF

ELSIF ((validProfileCounter+1) MOD 2 = 0)
THEN
  RETURN;
END_IF

// Find index of fastest Profile
Tmin := Constants.Infinity;
FOR i:=0 TO validProfileCounter
DO
  FOR j:=0 TO validProfileCounter
  DO
    IF validProfiles[i].t_sum[6] + validProfiles[i].Brake.Duration < validProfiles[j].t_sum[6] + validProfiles[j].Brake.Duration AND_THEN
       validProfiles[i].t_sum[6] + validProfiles[i].Brake.Duration < Tmin
    THEN
      Tmin := validProfiles[i].t_sum[6] + validProfiles[i].Brake.Duration + validProfiles[i].Accel.Duration;
      idx_min := i;
		END_IF
  END_FOR
END_FOR

